# B&R Automation Studio project RobotNewEra (part 9)

#### gmciplog.cnc
```
Root (LangModule=ailgcode, Version=1.0)
  AxesSpec
  PVMacros:
    DR8:
      REF = #next_motion.Data.R8_value
    DI4:
      REF = #next_motion.Data.I4_value
    DU4:
      REF = #next_motion.Data.UI4_value
    DR8_G211:
      SET = %_CNC.TA = ${EXPR};
       if (%_CNC.TA < 0)
         %_CNC.TA = 0;
       endif
        #next_motion.Data.R8_value = ${EXPR};
    Dlp:
      REF = #next_motion.Data.LinMovement.Position
    Dli:
      SET = #next_motion.Data.LinMovement.Idx[0] = ArrayRep(:(:-1:):);
        #next_motion.Data.LinMovement.Idx = ${EXPR};
    Dlm:
      SET = #next_motion.Data.LinMovement.Mode[0] = ArrayRep(:(:-1:):);
        #next_motion.Data.LinMovement.Mode = ${EXPR};
    Dto:
      REF = #next_motion.Data.Trans.Offset
    Dti:
      SET = #next_motion.Data.Trans.AxIdx[0] = ArrayRep(:(:-1:):);
        #next_motion.Data.Trans.AxIdx = ${EXPR};
    Dtm:
      SET = #next_motion.Data.Trans.Mode[0] = ArrayRep(:(:-1:):);
        #next_motion.Data.Trans.Mode = ${EXPR};
    Dcp:
      REF = #next_motion.Data.CircMovement.Parameter
    Dci:
      SET = #next_motion.Data.CircMovement.Idx[0] = ArrayRep(:(:-1:):);
        #next_motion.Data.CircMovement.Idx = ${EXPR};
    Dcm:
      SET = #next_motion.Data.CircMovement.Mode[0] = ArrayRep(:(:-1:):);
        #next_motion.Data.CircMovement.Mode = ${EXPR};
    Dtp:
      REF = #next_motion.Data.ToolAxOrient.Parameter
    Dts:
      REF = #next_motion.Data.ToolAxOrient.Sign
    Daz:
      REF = #next_motion.Data.AbsZeroPtShift.ZpRecIdx
    Dpt:
      SET = #next_motion.Data.ProgZeroPtShift.Type[0] = ArrayRep(:(:-1:):);
        #next_motion.Data.ProgZeroPtShift.Type = ${EXPR};
    Dpm:
      SET = #next_motion.Data.ProgZeroPtShift.Mode[0] = ArrayRep(:(:-1:):);
        #next_motion.Data.ProgZeroPtShift.Mode = ${EXPR};
    Dpa:
      REF = #next_motion.Data.ProgZeroPtShift.AxShift
    Dovpathdef:
      REF = #next_motion.Data.OptMotPar.path_definition
    Dovpathdefd:
      REF = #next_motion.Data.OptMotPar.path_definition_def
    Dorpar:
      REF = #next_motion.Data.OptMotPar.robot_par
    Dorpard:
      REF = #next_motion.Data.OptMotPar.robot_par_def
    Dolim:
      REF = #next_motion.Data.OptMotPar.limits_idx
    Dolimd:
      REF = #next_motion.Data.OptMotPar.limits_idx_def
    Dolimfac:
      REF = #next_motion.Data.OptMotPar.limits_factor
    Dolimfacd:
      REF = #next_motion.Data.OptMotPar.limits_factor_def
    Dfdx:
      REF = #next_motion.Data.FullTrfTool.Dx
    Dfdy:
      REF = #next_motion.Data.FullTrfTool.Dy
    Dfdz:
      REF = #next_motion.Data.FullTrfTool.Dz
    Dfph:
      REF = #next_motion.Data.FullTrfTool.Phi
    Dft:
      REF = #next_motion.Data.FullTrfTool.Theta
    Dfps:
      REF = #next_motion.Data.FullTrfTool.Psi
    DPLDli:
      REF = #next_motion.Data.PosLatchDistance.LatchIdx
    DPLDts:
      REF = #next_motion.Data.PosLatchDistance.TriggSource
    DPLDe:
      REF = #next_motion.Data.PosLatchDistance.Edge
    DPLDti:
      REF = #next_motion.Data.PosLatchDistance.HwTrigIdx
    DPLDd:
      REF = #next_motion.Data.PosLatchDistance.Distance
    DPLli:
      REF = #next_motion.Data.PosLatch.LatchIdx
    DPLts:
      REF = #next_motion.Data.PosLatch.TriggSource
    DPLe:
      REF = #next_motion.Data.PosLatch.Edge
    DPLti:
      REF = #next_motion.Data.PosLatch.HwTrigIdx
    Drma:
      REF = #next_motion.Data.R_DependFeed.MaxRadius
    Drmi:
      REF = #next_motion.Data.R_DependFeed.MinRadius
    Drr:
      REF = #next_motion.Data.R_DependFeed.Rate
    Dsvp:
      SET = #next_motion.Data.Set_v_jump.programmed[0] = ArrayRep(:(:ncOFF:):);
        #next_motion.Data.Set_v_jump.programmed = ${EXPR};
    Dsvv:
      REF = #next_motion.Data.Set_v_jump.value
    Dsap:
      SET = #next_motion.Data.Set_a_jump.programmed[0] = ArrayRep(:(:ncOFF:):);
        #next_motion.Data.Set_a_jump.programmed = ${EXPR};
    Dsav:
      REF = #next_motion.Data.Set_a_jump.value
    Dsep:
      SET = #next_motion.Data.SetAxLimit.programmed[0] = ArrayRep(:(:ncOFF:):);
        #next_motion.Data.SetAxLimit.programmed = ${EXPR};
    Dser:
      REF = #next_motion.Data.SetAxLimit.RecordIdx
    Dcad:
      REF = #next_motion.Data.CamWrapping.Diameter
    Dcap:
      REF = #next_motion.Data.CamWrapping.ParameterP1
    Dsu:
      REF = #next_motion.Data.SetPathAccDec.UnitType
    Dsv108:
      SET = #next_motion.Data.SetPathAccDec.value = ${EXPR};
        if (#next_motion.Data.SetPathAccDec.UnitType == 1)
          %_CNC.lim_path_acc_p = ${EXPR} / 100.0 * %_CNC.lim_path_acc_p_ini;
        else
          %_CNC.lim_path_acc_p = ${EXPR};
        endif
    Dsv109:
      SET = #next_motion.Data.SetPathAccDec.value = ${EXPR};
        if (#next_motion.Data.SetPathAccDec.UnitType == 1)
          %_CNC.lim_path_acc_n = ${EXPR} / 100.0 * %_CNC.lim_path_acc_n_ini;
        else
          %_CNC.lim_path_acc_n = ${EXPR};
        endif
    Dsv110:
      SET = #next_motion.Data.SetPathAccDec.value = ${EXPR};
        if (#next_motion.Data.SetPathAccDec.UnitType == 1)
          %_CNC.lim_path_acc_p = ${EXPR} / 100.0 * %_CNC.lim_path_acc_p_ini;
          %_CNC.lim_path_acc_n = ${EXPR} / 100.0 * %_CNC.lim_path_acc_n_ini;
        else
          %_CNC.lim_path_acc_p = ${EXPR};
          %_CNC.lim_path_acc_n = ${EXPR};
        endif
    Dsma:
      REF = #next_motion.Data.SetTransSpeed.MaxAngle
    Dsmi:
      REF = #next_motion.Data.SetTransSpeed.MinAngle
    Dsr:
      REF = #next_motion.Data.SetTransSpeed.RedFactor
    Dbrp:
      REF = #next_motion.Data.BezierSpline.RadiusProgrammed
    Dbr:
      REF = #next_motion.Data.BezierSpline.Radius
    Dbvp:
      REF = #next_motion.Data.BezierSpline.VeProgrammed
    Dbv:
      REF = #next_motion.Data.BezierSpline.Ve
    Dbl:
      REF = #next_motion.Data.BezierSpline.LinProgrammed
    Dbsf:
      REF = #next_motion.Data.BezierSpline.scalingFactor
    Dbsfd:
      REF = #next_motion.Data.BezierSpline.scalingFactor_def
    Dao:
      REF = #next_motion.Data.AutomTangentialAx.Offset
    Daa:
      REF = #next_motion.Data.AutomTangentialAx.AxIdx
    DAMa:
      REF = #next_motion.Data.AxisMapping.AxIdx
    DAMf:
      REF = #next_motion.Data.AxisMapping.factor
    DAMp:
      REF = #next_motion.Data.AxisMapping.ParameterP1
    DSPEt:
      REF = #next_motion.Data.SignalPathEnd.Time
    DSPEst:
      REF = #next_motion.Data.SignalPathEnd.SignalType
    DSPEsi:
      REF = #next_motion.Data.SignalPathEnd.SignalIdx
    DSPEsd:
      REF = #next_motion.Data.SignalPathEnd.SourceData
    DSPEd:
      REF = #next_motion.Data.SignalPathEnd.DataLength
    DSPEp:
      SET = #next_motion.Data.SignalPathEnd.pDestination = \#sys_vars.EXF[0];
    DSPEDst:
      REF = #next_motion.Data.SignalPathEndDist.SignalType
    DSPEDsi:
      REF = #next_motion.Data.SignalPathEndDist.SignalIdx
    DSPEDsd:
      REF = #next_motion.Data.SignalPathEndDist.SourceData
    DSPEDd:
      REF = #next_motion.Data.SignalPathEndDist.DataLength
    DSPEDp:
      SET = #next_motion.Data.SignalPathEndDist.pDestination = \#sys_vars.EXF[0];
    DSPo:
      REF = #next_motion.Data.SignalPredict.Override
    DWCx1:
      REF = #next_motion.Data.WS_Ctrl.x1
    DWCz1:
      REF = #next_motion.Data.WS_Ctrl.z1
    DWCy1:
      REF = #next_motion.Data.WS_Ctrl.y1
    DWCx2:
      REF = #next_motion.Data.WS_Ctrl.x2
    DWCz2:
      REF = #next_motion.Data.WS_Ctrl.y2
    DWCy2:
      REF = #next_motion.Data.WS_Ctrl.z2
    DWCi:
      REF = #next_motion.Data.WS_Ctrl.index
    DWCc:
      REF = #next_motion.Data.WS_Ctrl.coord
    DWCp:
      REF = #next_motion.Data.WS_Ctrl.pplane
    DWCo:
      REF = #next_motion.Data.WS_Ctrl.orient
    DWCs:
      REF = #next_motion.Data.WS_Ctrl.shape
    DWCa:
      SET = #next_motion.Data.WS_Ctrl.arm_diameter[0] = ArrayRep(:(:ncOFF:):);
        #next_motion.Data.WS_Ctrl.arm_diameter = ${EXPR};
    DTDRt:
      REF = #next_motion.Data.ToolDataRecord.ToolIdx
    Sz:
      REF = #sys_vars.ZP
    DSSi:
      REF = #next_motion.Data.SpindleSpeed.Idx
    DSSs:
      REF = #next_motion.Data.SpindleSpeed.speed
    DCSSt:
      REF = #next_motion.Data.C2_SplineStart.BCType
    DCSSv:
      REF = #next_motion.Data.C2_SplineStart.BCValue
    DCSSp:
      SET = #next_motion.Data.C2_SplineStart.BCProgrammed[0] = ArrayRep(:(:ncOFF:):);
        #next_motion.Data.C2_SplineStart.BCProgrammed = ${EXPR};
    DCSSsp:
      REF = #next_motion.Data.C2_SplineStart.SegmentParameter
    DCSSst:
      REF = #next_motion.Data.C2_SplineStart.SegmentType
    DCSEt:
      REF = #next_motion.Data.C2_SplineEnd.BCType
    DCSEv:
      REF = #next_motion.Data.C2_SplineEnd.BCValue
    DCSEp:
      SET = #next_motion.Data.C2_SplineEnd.BCProgrammed[0] = ArrayRep(:(:ncOFF:):);
        #next_motion.Data.C2_SplineEnd.BCProgrammed = ${EXPR};
    DFd:
      REF = #next_motion.Data.Frame.Data
    DSVs:
      REF = #next_motion.Data.SystemVariable.SysVarIdx
    DSVa:
      REF = #next_motion.Data.SystemVariable.AxIdx
    DSVd:
      REF = #next_motion.Data.SystemVariable.Data.R8_value
    DABNf:
      REF = #next_motion.Data.AutoBlockNumber.offset
    DABNo:
      REF = #next_motion.Data.AutoBlockNumber.factor
    DCSSPs:
      REF = #next_motion.Data.ConstantSurfaceSpeed.Speed
    DCSSPp:
      REF = #next_motion.Data.ConstantSurfaceSpeed.Programmed
    MXFPx:
      REF = #next_motion.Data.MXFrame.Pos.x
    MXFPy:
      REF = #next_motion.Data.MXFrame.Pos.y
    MXFPz:
      REF = #next_motion.Data.MXFrame.Pos.z
    MXFOt:
      REF = #next_motion.Data.MXFrame.Orient.Type
    MXFOa:
      REF = #next_motion.Data.MXFrame.Orient.Angle
    MXTFPx:
      REF = #next_motion.Data.MXTool.Frame.Pos.x
    MXTFPy:
      REF = #next_motion.Data.MXTool.Frame.Pos.y
    MXTFPz:
      REF = #next_motion.Data.MXTool.Frame.Pos.z
    MXTFOt:
      REF = #next_motion.Data.MXTool.Frame.Orient.Type
    MXTFOa:
      REF = #next_motion.Data.MXTool.Frame.Orient.Angle
    MXTr:
      REF = #next_motion.Data.MXTool.Radius
    MXPPx:
      REF = #next_motion.Data.MXPoint.Pos.x
    MXPPy:
      REF = #next_motion.Data.MXPoint.Pos.y
    MXPPz:
      REF = #next_motion.Data.MXPoint.Pos.z
    MXPOt:
      REF = #next_motion.Data.MXPoint.Orient.Type
    MXPOa:
      REF = #next_motion.Data.MXPoint.Orient.Angle
    MXPCm:
      REF = #next_motion.Data.MXPoint.Cfg.Mode
    MXPr:
      REF = #next_motion.Data.MXPoint.RotAxis
    MXPa:
      REF = #next_motion.Data.MXPoint.AuxAxis
    MXPhTr:
      REF = #next_motion.Data.MXPathDesc.Trans.Radius
    MXPhTt:
      REF = #next_motion.Data.MXPathDesc.Trans.Type
    MXDa:
      REF = #next_motion.Data.MXDynamicDesc.Accel
    MXDd:
      REF = #next_motion.Data.MXDynamicDesc.Decel
    MXDOe:
      REF = #next_motion.Data.MXDynamicDesc.Optmot.Enable
    MXDOv:
      REF = #next_motion.Data.MXDynamicDesc.Optmot.VelPathDef
    MXDOr:
      REF = #next_motion.Data.MXDynamicDesc.Optmot.RobotPar
    MXDOl:
      REF = #next_motion.Data.MXDynamicDesc.Optmot.Limits
    MXVv:
      REF = #next_motion.Data.MXVelocity.v
    MXVm:
      REF = #next_motion.Data.MXVelocity.Mode
    MXAj:
      REF = #next_motion.Data.MXAxisTarget.JointAxis
    MXAa:
      REF = #next_motion.Data.MXAxisTarget.AuxAxis
    MXAb:
      REF = #next_motion.Data.MXAxisTarget.BaseAxis
    MXJ:
      REF = #next_motion.Data.MXJointAxis
    MXAto:
      REF = #next_motion.Data.MXAutoTang.Offset
    MXCDCas:
      REF = #next_motion.Data.MXCDC.ArcTransSpd
    MXCDCsm:
      REF = #next_motion.Data.MXCDC.SpdMode
    MXCDCcv:
      REF = #next_motion.Data.MXCDC.ContourViolation
    MXCDCtm:
      REF = #next_motion.Data.MXCDC.TransMode
    MXCDCem:
      REF = #next_motion.Data.MXCDC.EntryMode
    MXCDCal:
      REF = #next_motion.Data.MXCDC.AcrToLine
    THCp:
      REF = #next_motion.Data.ThreadCut.Position
    THCi:
      SET = #next_motion.Data.ThreadCut.Idx[0] = ArrayRep(:(:-1:):);
        #next_motion.Data.ThreadCut.Idx = ${EXPR};
    THCm:
      SET = #next_motion.Data.ThreadCut.Mode[0] = ArrayRep(:(:-1:):);
        #next_motion.Data.ThreadCut.Mode = ${EXPR};
    THCld:
      REF = #next_motion.Data.ThreadCut.LeadDirection
    THCl:
      REF = #next_motion.Data.ThreadCut.Lead
    THCo:
      REF = #next_motion.Data.ThreadCut.Offset
    ACVc:
      REF = #next_motion.Data.AxisCtrlVelocity.Command
    ACVi:
      REF = #next_motion.Data.AxisCtrlVelocity.Idx
    ACSs:
      REF = #next_motion.Data.AxisCtrlSpeed.Speed
    ACSi:
      REF = #next_motion.Data.AxisCtrlSpeed.Idx
    ACPp:
      REF = #next_motion.Data.AxisCtrlPosition.Position
    ACPd:
      REF = #next_motion.Data.AxisCtrlPosition.PositionDefined
    ACPi:
      REF = #next_motion.Data.AxisCtrlPosition.Idx
    ACPm:
      REF = #next_motion.Data.AxisCtrlPosition.Mode
    CHFm:
      REF = #next_motion.Data.Champfer.Mode
    CHFv:
      REF = #next_motion.Data.Champfer.Value
    GENd:
      REF = #next_motion.Data.GenericData.Data
  Constants:
    PathBusy = BUSY (type=STRING)
    PathStatus = STATUS (type=STRING)
    PathErrLevel = ERRLEV (type=STRING)
  BuiltInProcs:
    SendCommand = SendCommand(:$[1]:); (MinArgs=1, MaxArgs=1, Inline=Yes)
    DispatchAndWait = DispatchAndWait(:$[1]:); (MinArgs=1, MaxArgs=1, Inline=Yes)
  Preprocess:
    MP_PJN (Search=MP22000 , Replace=PJN )
    MP_PJB (Search=MP22100 , Replace=PJB )
  GCodes:
    G_DELAY (GNum=0, Alias=@, AliasIsPattern=Yes, Inline=Yes)
      Arg (DataType=FLOAT, ref=tickdelay)
    G_PJN (GNum=22000, Alias=PJN, Inline=Yes, Group=220)
      Arg PathBusy (DataType=FLOAT, ref=busy_count)
      Arg PathStatus (DataType=FLOAT, ref=final_status)
      Arg PathErrLevel (DataType=FLOAT, ref=error_level)
    G_PJB (GNum=22100, Alias=PJB, Inline=Yes, Group=220)
      Arg PathBusy (DataType=FLOAT, ref=busy_count)
      Arg PathStatus (DataType=FLOAT, ref=final_status)
      Arg PathErrLevel (DataType=FLOAT, ref=error_level)
  MCodes:
    M_DEFAULT (IsDefault=Yes, MinValue=0, MaxValue=999999)
      ARG (ref=VALUE, DataType=FLOAT, RequireLiteral=Yes)
    M10003 = 10003 (Inline=Yes)
      ARG (ref=VALUE, DataType=FLOAT, RequireLiteral=Yes)
    M1000000 = 1000000 (Alias=;, AliasIsPattern=Yes, Inline=Yes, IgnoreIfGroups=220)
      ARG (ref=VALUE, DataType=FLOAT, RequireLiteral=Yes)
  ParserData (NestedComments=No, DefaultCaseSensitive=Yes, CommentsSpanLines=No, ReadWholeFileBeforeParsing=No, ExpectMainProgStmts=Yes, UseFubTemplates=No)
    TKG_END_OF_LINE = \n (IsPattern=No)
    TKG_OPEN_COMMENT = #
    TKG_NC_BLOCK_PREFIX = N:[\s\d] (IsPattern=Yes)
    TKG_OPEN_LISTBRACKET = (
    TKG_CLOSE_LISTBRACKET = )
    TKG_COMMA = ,
    TKG_NUMBER = \d+\.\d+|\d+\.|\.\d+ (IsPattern=Yes)
    TKG_INTEGER = \d+ (IsPattern=Yes)
    TKG_NUMBER_EXP = e:[\s\d\+\-\.] (IsPattern=Yes)
    TKG_ASSIGN_EQ = =
    TKG_ARITH_BINARY_MINUS = -
    TKG_M_CODE_PREFIX = MP:\d (IsPattern=Yes)
  StringChars (AsciiStringStart=")
    EscapeSeq (Search=$N, CaseSensitive=No, ReplaceValue=10)
    EscapeSeq (Search=$L, CaseSensitive=Yes, ReplaceValue=10)
    EscapeSeq (Search=$Q, CaseSensitive=No, ReplaceStr=")
    EscapeSeq (Search=$[\dA-F]+, IsPattern=Yes, CaseSensitive=No, ReplaceEncodingBase=16)
    EscapeSeq (Search=$$, ReplaceStr=$)
    EscapeSeq (Search=$, ReplaceStr=)
```

- Data object Logical/MotionHandling/Interpreter/GmcIpConfig/gmcipesm (Cnc, version 2.47.4) (no source held here)

### Data object Logical/MotionHandling/Interpreter/GmcIpConfig/gmcipmxd (Cnc, version 2.47.4)

#### gmcipmxd.cnc
```
(********************************************************************
 * COPYRIGHT -- Bernecker + Rainer
 ********************************************************************
 * Library: Motion Command Extension
 * File: arnc0mx.typ
 * Author: B&R
 ********************************************************************
 * Data types of Motion Command Library
 ********************************************************************)

TYPE
	MXOrientationType : STRUCT
		Type : UDINT;
		Angle : ARRAY[0..3]OF LREAL;
	END_STRUCT;
	MXPositionType : STRUCT
		x : LREAL;
		y : LREAL;
		z : LREAL;
	END_STRUCT;
	MXFrameType : 	STRUCT
		Pos : MXPositionType;
		Orient : MXOrientationType;
	END_STRUCT;
	MXToolType : STRUCT
		Frame : MXFrameType;
		Radius : LREAL;
	END_STRUCT;
	MXJointAxisType :ARRAY[0..5]OF LREAL;
	MXAuxAxisType :ARRAY[0..14]OF LREAL;
	MXBaseAxisType :ARRAY[0..5]OF LREAL;
	MXRotAxisType :ARRAY[0..5]OF LREAL;
	MXConfigType : 	STRUCT
		Mode : UDINT;
	END_STRUCT;
	MXPointType : 	STRUCT
		Pos : MXPositionType;
		Orient : MXOrientationType;
		Cfg : MXConfigType;
		RotAxis : MXRotAxisType;
		AuxAxis : MXAuxAxisType;
	END_STRUCT;
	MXPathTransType : STRUCT
		Radius	:	LREAL;
		Type	:	UDINT;
	END_STRUCT;
	MXPathDescType : STRUCT
		Trans	:	MXPathTransType;
	END_STRUCT;
	MXOptMotType : STRUCT
		Enable : BOOL;
		VelPathDef : USINT;
		RobotPar : USINT;
		Limits : USINT;
	END_STRUCT;
	MXDynamicDescType :	STRUCT
		Accel : LREAL := 100;
		Decel : LREAL := 100;
		Optmot : MXOptMotType;
	END_STRUCT;
	MXHWTrigType : 	STRUCT
		Source : USINT;
		Index : USINT;
	END_STRUCT;
	MXSWTrigType : STRUCT
		Expression : STRING[64];
	END_STRUCT;
	MXTriggConfigType :	STRUCT
		Type : UINT;
		HWTrig : MXHWTrigType;
		SWTrig : MXSWTrigType;
		Edge : USINT;
		ResidPath : USINT;
	END_STRUCT;
	MXVelocityType : STRUCT
		v : LREAL;
		Mode : UDINT := 1;
	END_STRUCT;
	MXAxisTargetType : 	STRUCT
		JointAxis : MXJointAxisType;
		AuxAxis : MXAuxAxisType;
		BaseAxis : MXBaseAxisType;
	END_STRUCT;
	MXCDCType : STRUCT
		ArcTransSpd : LREAL := 100;
		SpdMode : UDINT;
		ContourViolation : UDINT;
		TransMode : UDINT;
		EntryMode : USINT;
		AcrToLine : BOOL;
	END_STRUCT;
	MXAutoTangType : STRUCT
		Offset : LREAL;
	END_STRUCT;
	MXHWTriggerType :	STRUCT
		Source : UINT;
		Index : UINT;
	END_STRUCT;
	MXTriggerConfigType : 	STRUCT
		Type : UINT;
		Edge : UINT;
		HWTrigger : MXHWTriggerType;
	END_STRUCT;
END_TYPE

(********************************************************************
 * COPYRIGHT (C) BERNECKER + RAINER, AUSTRIA, A-5142 EGGELSBERG
 ********************************************************************
 * Library: ARNC0MX
 * File: arnc0mx.fun
 * Created: 13.06.2012
 ********************************************************************
 * Functions and function blocks of library ARNC0MX
 ********************************************************************)
FUNCTION MXPointToJointEx1 : UDINT
	VAR_INPUT
		AddrTrfData : UDINT;
		Point : MXPointType;
		Joint : MXJointAxisType;
		TrfType : UDINT;
		Tool : MXToolType;
		BaseFrame : MXFrameType;
		RefJoint : ARRAY[0..5] OF LREAL;
	END_VAR
END_FUNCTION

FUNCTION MXPointToJointEx : UDINT
	VAR_INPUT
		AddrTrfData : UDINT;
		Point : MXPointType;
		Joint : MXJointAxisType;
		TrfType : UDINT;
		Tool : MXToolType;
		BaseFrame : MXFrameType;
		RefJoint : MXJointAxisType;
	END_VAR
END_FUNCTION

FUNCTION MXJointToPointEx1 : UDINT
	VAR_INPUT
		AddrTrfData : UDINT;
		Joint : MXJointAxisType;
		Point : MXPointType;
		AnglesType : UDINT;
		TrfType : UDINT;
		Tool : MXToolType;
		BaseFrame : MXFrameType;
		RefPath : ARRAY[0..5] OF LREAL;
	END_VAR
END_FUNCTION

FUNCTION MXJointToPointEx : UDINT
	VAR_INPUT
		AddrTrfData : UDINT;
		Joint : MXJointAxisType;
		Point : MXPointType;
		AnglesType : UDINT;
		TrfType : UDINT;
		Tool : MXToolType;
		BaseFrame : MXFrameType;
		RefPoint : MXPointType;
	END_VAR
END_FUNCTION

FUNCTION MXCncAxesToPoint : UDINT
	VAR_INPUT
		AddrTrfData : UDINT;
		Axis : ARRAY[0..14] OF LREAL;
		Point : MXPointType;
		TrfType : UDINT;
		AnglesType : UDINT;
		AxisMapCode : ARRAY[0..14] OF UINT;
		AxisMapIdx : ARRAY[0..14] OF UINT;
		ActiveAxesCount : UDINT;
	END_VAR
END_FUNCTION

FUNCTION MXFromOrient : UDINT
	VAR_INPUT
		Orient : MXOrientationType;
		Matrix : ARRAY[0..8] OF LREAL;
	END_VAR
END_FUNCTION

FUNCTION MXToOrient : UDINT
	VAR_INPUT
		Matrix : ARRAY[0..8] OF LREAL;
		Type : UDINT;
		Orient : MXOrientationType;
		RefAngle : ARRAY[0..2] OF LREAL;
	END_VAR
END_FUNCTION

FUNCTION MXConvertOrient : UDINT
	VAR_INPUT
		OrientIn : MXOrientationType;
		Type : UDINT;
		OrientOut : MXOrientationType;
		RefAngle : ARRAY[0..2] OF LREAL;
	END_VAR
END_FUNCTION

FUNCTION MXFrameRotX : UDINT
	VAR_INPUT
		Frame : MXFrameType;
		Angle : LREAL;
	END_VAR
END_FUNCTION

FUNCTION MXFrameRotY : UDINT
	VAR_INPUT
		Frame : MXFrameType;
		Angle : LREAL;
	END_VAR
END_FUNCTION

FUNCTION MXFrameRotZ : UDINT
	VAR_INPUT
		Frame : MXFrameType;
		Angle : LREAL;
	END_VAR
END_FUNCTION

FUNCTION MXFrameEuler : UDINT
	VAR_INPUT
		Frame : MXFrameType;
		Phi : LREAL;
		Theta : LREAL;
		Psi : LREAL;
	END_VAR
END_FUNCTION

FUNCTION MXFrameRPY : UDINT
	VAR_INPUT
		Frame : MXFrameType;
		Roll : LREAL;
		Pitch : LREAL;
		Yaw : LREAL;
	END_VAR
END_FUNCTION

FUNCTION MXFrameTrans : UDINT
	VAR_INPUT
		Frame : MXFrameType;
		DistanceX : LREAL;
		DistanceY : LREAL;
		DistanceZ : LREAL;
	END_VAR
END_FUNCTION

FUNCTION MXFrameTransX : UDINT
	VAR_INPUT
		Frame : MXFrameType;
		Distance : LREAL;
	END_VAR
END_FUNCTION

FUNCTION MXFrameTransY : UDINT
	VAR_INPUT
		Frame : MXFrameType;
		Distance : LREAL;
	END_VAR
END_FUNCTION

FUNCTION MXFrameTransZ : UDINT
	VAR_INPUT
		Frame : MXFrameType;
		Distance : LREAL;
	END_VAR
END_FUNCTION

FUNCTION MXFrameApply : UDINT
	VAR_INPUT
		Frame1 : MXFrameType;
		Frame2 : MXFrameType;
	END_VAR
END_FUNCTION

FUNCTION MXFromFrame : UDINT
	VAR_INPUT
		Frame : MXFrameType;
		PointIn : MXPointType;
		PointOut : MXPointType;
	END_VAR
END_FUNCTION

FUNCTION MXToFrame : UDINT
	VAR_INPUT
		Frame : MXFrameType;
		PointIn : MXPointType;
		PointOut : MXPointType;
	END_VAR
END_FUNCTION

(********************************************************************
 * COPYRIGHT -- Bernecker + Rainer
 ********************************************************************
 * Library: Motion Command Extension
 * File: arnc0mx.var
 * Author: B&R
 ********************************************************************
 * Constants of Motion Command Library
 ********************************************************************)

(* Velocity mode constants (<MXVelocityType>.Mode) *)
VAR CONSTANT
  MX_VEL_MODE_RAPID : UDINT := 0; (* rapid mode *)
  MX_VEL_MODE_FEED  : UDINT := 1; (* feedrate mode *)
  MX_VEL_MODE_TIME  : UDINT := 2; (* inverse time mode *)
END_VAR

(* MXVelocityType constants *)
VAR CONSTANT
  MX_VEL_RAPID  : MXVelocityType := (Mode:=0);           (* rapid movement         *)
  MX_VEL_F50000 : MXVelocityType := (v:=50000, Mode:=1); (* 50000 units per minute *)
  MX_VEL_F10000 : MXVelocityType := (v:=10000, Mode:=1); (* 10000 units per minute *)
  MX_VEL_F5000  : MXVelocityType := (v:=5000,  Mode:=1); (* 5000 units per minute  *)
  MX_VEL_F1000  : MXVelocityType := (v:=1000,  Mode:=1); (* 1000 units per minute  *)
  MX_VEL_F500   : MXVelocityType := (v:=500,   Mode:=1); (* 500 units per minute   *)
  MX_VEL_F100   : MXVelocityType := (v:=100,   Mode:=1); (* 100 units per minute   *)
END_VAR

(* Trigger configuration constants *)
VAR CONSTANT
  MX_TRIGGER_HW	            : UINT := 0;           (* Hardware trigger - MXHWTriggerType *)
  MX_TRIGGER_POSITIVE_EDGE  : UINT := 0;           (* Positive edge						 *)
  MX_TRIGGER_NEGATIVE_EDGE  : UINT := 1;           (* Negative edge						 *)
  MX_TRIGGER_HW_INPUT1		: UINT := 1;           (* Hardware trigger input 1			 *)
  MX_TRIGGER_HW_INPUT2		: UINT := 2;           (* Hardware trigger input 1			 *)
END_VAR

(* MXFrameMXFrameType constants *)
VAR CONSTANT
  MX_FRM_ZERO : MXFrameType := (0); (* zero (identity) frame *)
END_VAR

(* Transition type constants (<MXPathTransType>.Type) *)
VAR CONSTANT
  MX_TRANS_OFF      : UDINT := 0; (* Transition deactivated *)
  MX_TRANS_ACCURATE : UDINT := 1; (* Accuracy hold *)
  MX_TRANS_ARC      : UDINT := 2; (* Tangential transition arcs *)
  MX_TRANS_ROUND    : UDINT := 3; (* Rounding edges *)
END_VAR

(* Orientation type constants (<MXOrientationType>.Type) matches constants from TRF_LIB *)
VAR CONSTANT
  MX_CARDAN_XYZ_ANGLES    : UDINT := 1;      (* Cardan XYZ angles *)
  MX_EULER_XYZ_ANGLES     : UDINT := 1;      (* Cardan XYZ angles *)
  MX_CARDAN_XZY_ANGLES    : UDINT := 2;      (* Cardan XZY angles *)
  MX_EULER_XZY_ANGLES     : UDINT := 2;      (* Cardan XZY angles *)
  MX_CARDAN_YXZ_ANGLES    : UDINT := 4;      (* Cardan YXZ angles *)
  MX_EULER_YXZ_ANGLES     : UDINT := 4;      (* Cardan YXZ angles *)
  MX_CARDAN_YZX_ANGLES    : UDINT := 8;      (* Cardan YZX angles *)
  MX_EULER_YZX_ANGLES     : UDINT := 8;      (* Cardan YZX angles *)
  MX_CARDAN_ZXY_ANGLES    : UDINT := 16;     (* Cardan ZXY angles *)
  MX_EULER_ZXY_ANGLES     : UDINT := 16;     (* Cardan ZXY angles *)
  MX_CARDAN_ZYX_ANGLES    : UDINT := 32;     (* Cardan ZYX angles *)
  MX_EULER_ZYX_ANGLES     : UDINT := 32;     (* Cardan ZYX angles *)
  MX_EULER_XYX_ANGLES     : UDINT := 64;     (* Euler XYX angles  *)
  MX_EULER_XZX_ANGLES     : UDINT := 128;    (* Euler XZX angles  *)
  MX_EULER_YXY_ANGLES     : UDINT := 256;    (* Euler YXY angles  *)
  MX_EULER_YZY_ANGLES     : UDINT := 512;    (* Euler YZY angles  *)
  MX_EULER_ZXZ_ANGLES     : UDINT := 1024;   (* Euler ZXZ angles  *)
  MX_EULER_ZYZ_ANGLES     : UDINT := 2048;   (* Euler ZYZ angles  *)
  MX_POSITIVE_ANGLES      : UDINT := 4096;   (* mathematically positive angles *)
  MX_NEGATIVE_ANGLES      : UDINT := 8192;   (* mathematically negative angles *)
  MX_DIRECT_ANGLES        : UDINT := 16384;  (* direct "R" rotation matrix     *)
  MX_INDIRECT_ANGLES      : UDINT := 32768;  (* indirect "R^T" rotation matrix *)
  MX_EULER_ANGLES         : UDINT := 1024;   (* Euler ZXZ is commonly in view  *)
  MX_CARDAN_ANGLES        : UDINT := 1;      (* Cardan XYZ is commonly in view *)
  MX_NAUTICAL_ANGLES      : UDINT := 1;      (* Cardan XYZ is commonly in view *)
  MX_TAIT_BRYAN_ANGLES    : UDINT := 1;      (* Cardan XYZ is commonly in view *)
  MX_QUATERNION           : UDINT := 8000;   (* quaternion *)
END_VAR

(* Kinematics configuration mode constants (<MXConfigType>.Mode) matches constants from TRF_LIB *)
VAR CONSTANT
  MX_MODE_FRONT           : UDINT := 1;          (* front *)
  MX_MODE_BACK            : UDINT := 2;          (* back *)
  MX_MODE_CONVEX          : UDINT := 4;          (* convex *)
  MX_MODE_CONCAVE         : UDINT := 8;          (* concave *)
  MX_MODE_POSITIVE        : UDINT := 16;         (* positive *)
  MX_MODE_NEGATIVE        : UDINT := 32;         (* negative *)
  MX_MODE_LEFT            : UDINT := 64;         (* left *)
  MX_MODE_RIGHT           : UDINT := 128;        (* right *)
  MX_MODE_DIRECT          : UDINT := 256;        (* direct *)
  MX_MODE_INDIRECT        : UDINT := 512;        (* indirect *)
  MX_MODE_CONVEX2         : UDINT := 1024;       (* convex2 *)
  MX_MODE_CONCAVE2        : UDINT := 2048;       (* concave2 *)
  MX_MODE_CONVEX3         : UDINT := 4096;       (* convex3 *)
  MX_MODE_CONCAVE3        : UDINT := 8192;       (* concave3 *)
  MX_MODE_HETEROGENEOUS   : UDINT := 16384;      (* heterogeneous *)
  MX_MODE_HOMOGENEOUS     : UDINT := 32768;      (* homogeneous *)
  MX_MODE_LEFT2           : UDINT := 65536;      (* left2 *)
  MX_MODE_RIGHT2          : UDINT := 131072;     (* right2 *)
  MX_MODE_NEG_DIR         : UDINT := 268435456;  (* negative direction forced *)
  MX_MODE_POS_DIR         : UDINT := 536870912;  (* positive direction forced *)
  MX_MODE_IN_SW_ENDS      : UDINT := 1073741824; (* in SW ends *)
END_VAR

(* Cutter diameter compensation constants *)
VAR CONSTANT
  MX_CDC_LEFT                    : UDINT := 0;      (* CDC left *)
  MX_CDC_RIGHT                   : UDINT := 1;      (* CDC right *)
  MX_CDC_SPD_ON_CONTOUR          : UDINT := 0;      (* Path speed moves to the contour *)
  MX_CDC_SPD_ON_TCP              : UDINT := 1;      (* Path speed moves to the center of the tool *)
  MX_CDC_NO_COUNTER_VIOLATION    : UDINT := 0;      (* Do NOT allow contour violations due to very short path *)
  MX_CDC_VIOLATION_SHORT_PATH    : UDINT := 1;      (* Allow contour violations due to very short path sections *)
  MX_CDC_VIOLATION_INNER_EDGE    : UDINT := 2;      (* Allow contour violations due to an inner edge without intersection *)
  MX_CDC_LINEAR_TRANSITION       : UDINT := 0;      (* CDC with linear transitions *)
  MX_CDC_ARC_TRANSITION          : UDINT := 1;      (* CDC with arc transitions *)
  MX_CDC_ENTRY_BLOCK             : UDINT := 0;      (* Activate/deactivate CDC indirectly with transi-tion block *)
  MX_CDC_ENTRY_DIRECT            : UDINT := 1;      (* Activate/deactivate CDC directly *)
  MX_CDC_ENTRY_INDIRECT          : UDINT := 2;      (* Activate/deactivate CDC indirectly *)
  MX_CDC_NO_ARC_TO_LINE          : UDINT := 0;      (* Deactivate replacement of arc with straight line *)
  MX_CDC_ARC_TO_LINE             : UDINT := 1;      (* Activate replacement of arc with straight line *)
END_VAR

(* Transformation function types *)
VAR CONSTANT
  MX_TRF_TYPE_INVERSE            : UDINT := 0;      (* TRF_inverse  function *)
  MX_TRF_TYPE_INVERSE2           : UDINT := 1;      (* TRF_inverse2 function *)
  MX_TRF_TYPE_INVERSE3           : UDINT := 2;      (* TRF_inverse3 function *)
  MX_TRF_TYPE_DIRECT             : UDINT := 0;      (* TRF_direct   function *)
  MX_TRF_TYPE_DIRECT2            : UDINT := 1;      (* TRF_direct2  function *)
  MX_TRF_TYPE_DIRECT3            : UDINT := 2;      (* TRF_direct3  function *)
END_VAR

(* Statuses, warnings, errors *)
VAR CONSTANT
  MX_OK                          : UDINT := 0;     (* Status OK *)
  MX_WARNING_AXES                : UDINT := 2001;  (* Transformation returns valid values with warnings on axes *)
  MX_WARNING_REF_POINT_ANGLES    : UDINT := 2002;  (* Values in reference point or reference joint axes may be ignored due to conversion to another angles type *)
  MX_ERROR_WRONG_ANGLE_TYPE      : UDINT := 6001;  (* Angles type is not supported *)
  MX_ERROR_TRF_DATA_NOT_DEFINED  : UDINT := 6002;  (* Address of the transformation data variable is zero *)
  MX_ERROR_WRONG_ROBOT           : UDINT := 6003;  (* Robot is not supported *)
  MX_ERROR_WRONG_TRF_TYPE        : UDINT := 6004;  (* Transformation type not supported *)
  MX_ERROR_TRF_LIB_NOT_SUPPORTED : UDINT := 6005;  (* Transformation library of not supported version *)
  MX_ERROR_TRF_CMD_CODE			 : UDINT := 8001;  (* Unknown command code *)
  MX_ERROR_TRF_MEASURE           : UDINT := 8002;  (* Unknown measure *)
  MX_ERROR_TRF_ANGLES_TYPE       : UDINT := 8003;  (* Unknown angles type *)
  MX_ERROR_TRF_GEN29_CMD_CODE    : UDINT := 9001;  (* Unknown command code *)
  MX_ERROR_UNKNOWN_ROBOT         : UDINT := 9002;  (* Unknown robot *)
  MX_ERROR_INVALID_TRF_TYPE      : UDINT := 9003;  (* Invalid type of transformation *)
  MX_ERROR_TRF_ERROR_AXES        : UDINT := 10003; (* Transformation function returns error of axis *)
  MX_ERROR_TRF_NOT_LICENSED      : UDINT := 10008; (* Transformation function not licenced *)
  MX_ERROR_TRF_NOT_SUPPORTED     : UDINT := 10009; (* Transformation function not supported *)
  MX_ERROR_FCT_NOT_DEFINED       : UDINT := 10010; (* Transformation function address is zero *)
  MX_ERROR_TRF_INVALID_INPUTS    : UDINT := 10015; (* Invalid inputs for transformation error *)
END_VAR

(* Error offsets *)
VAR CONSTANT
  MX_OFFSET_WARNING              : UDINT := 2000;  (* ARNC0MX warnings *)
  MX_OFFSET_WARNING_TRF_FUN      : UDINT := 4000;  (* TRF_LIB warnings *)
  MX_OFFSET_ERROR                : UDINT := 6000;  (* ARNC0MX errros *)
  MX_OFFSET_ERROR_TRF_FUN        : UDINT := 12000; (* TRF_LIB errors *)
END_VAR

(********************************************************************
 * COPYRIGHT -- Bernecker + Rainer
 ********************************************************************
 * Library: Motion Command Library
 * File: arnc0mxsv.var
 * Author: B&R
 ********************************************************************
 * System Variables of Motion Command Library
 ********************************************************************)
VAR {SHARED_IP_GLOBAL}
   _Frm  : MXFrameType;
   _Tool : MXToolType;
   _Vel  : MXVelocityType;
   _Base : MXFrameType;
   _Ref  : MXJointAxisType;
   _Pth  : MXPathDescType;
   _Dyn  : MXDynamicDescType;
END_VAR

VAR CONSTANT
   FRM_0   : MXFrameType := (0);
   POINT_0 : MXPointType := (0);
   BASE_0  : MXFrameType := (0);
   TOOL_0  : MXToolType  := (0);
   VEL_0   : MXVelocityType := (v:= 10000, Mode:=1); (* Default Feedrate = 10000*)
   REF_0   : MXJointAxisType := (0);
   VEC6_0  : ARRAY[0..5] OF LREAL := 6(0.0);
   PTH_0   : MXPathDescType := (0);
   DYN_0   : MXDynamicDescType := (Optmot:=(Enable:=1));
   AXIS_TARGET_0 : MXAxisTargetType := (0);
END_VAR

VAR {SHARED_IP_GLOBAL}
  __tmp_point : MXPointType;
  __tmp_frame : MXFrameType;
  __tmp_tool : MXToolType;
  __tmp_vel : MXVelocityType;
  __tmp_joint_axis : MXJointAxisType;
  __tmp_axis_target : MXAxisTargetType;
  __tmp_pth : MXPathDescType;
  __tmp_dynamic : MXDynamicDescType;
  __tmp_cdc : MXCDCType;
  __tmp_auto_tang : MXAutoTangType;
  __tmp_trigger : MXTriggerConfigType;
  __mx_status : UDINT;
  __tmp_vec6 : ARRAY[0..5] OF LREAL;
  __tmp_set_pos : ARRAY[0..14] OF LREAL;
  __tmp_axis_code : ARRAY[0..14] OF UINT;
  __tmp_axis_idx : ARRAY[0..14] OF UINT;
END_VAR
```

### Data object Logical/MotionHandling/Interpreter/GmcIpConfig/gmcipmx (Cnc, version 2.47.4)

#### gmcipmx.cnc
```
Root (LangModule=ailgcode, Version=1.0)
  AILHeader = sub OnProgStart
      %_Frm = %FRM_0;
      %_Base = %BASE_0;
      %_Tool = %TOOL_0;
      %_Vel = %VEL_0;
      %_Pth = %PTH_0;
      %_Dyn = %DYN_0;
      BlockCpy(:\%_Ref, \%REF_0:);
    endsub    
    
	sub OnProgEnd
	  #next_motion.Command = MPCMD_SEGMENTATION_END;
      PushPacket(::);
	endsub
  BuiltInProcs:
    WAIT_PP_SYNC = #next_motion.Command = MPCMD_IP_SYNCH_PP;
      PushPacket(::);
      DispatchAndWait(:IPCMD_SYNC_PP_CONT:);
    ERROR_EX = ErrorEx(:"id":$[1],"fmt":$[2],"data":(:$[3],$[4],$[5],$[6],$[7],$[8],$[9],$[10],$[11],$[12],$[13],$[14]:):); (MinArgs=3, MaxArgs=14)
    SET_POINT:
      Arg (ref=POINT, DataType=ANY_DATA, MinCount=1, MaxCount=1)
    SET_TRIGGER_CONFIG:
      Arg (ref=TRIGGER, DataType=ANY_DATA, MinCount=1, MaxCount=1)
      Arg (ref=bHALT, DataType=ANY_DATA, MinCount=1, MaxCount=1)
      Arg (ref=ID, DataType=ANY_DATA, MinCount=1, MaxCount=1)
    SET_WANTED_JOINT:
      Arg (ref=Ref, DataType=ANY_DATA, MinCount=1, MaxCount=1)
    SET_CIRCLE:
      Arg (ref=END_POINT, DataType=ANY_DATA, MinCount=1, MaxCount=1)
      Arg (ref=CIRCLE_POINT, DataType=ANY_DATA, MinCount=1, MaxCount=1)
    SET_AXIS_TARGET:
      Arg (ref=AXIS_TARGET, DataType=ANY_DATA, MinCount=1, MaxCount=1)
    SET_FRAME:
      Arg (ref=Frm, DataType=ANY_DATA, MinCount=0, MaxCount=1)
    SET_BASEFRAME:
      Arg (ref=Base, DataType=ANY_DATA, MinCount=0, MaxCount=1)
    SET_TOOL:
      Arg (ref=Tool, DataType=ANY_DATA, MinCount=0, MaxCount=1)
    SET_PATH_DESC:
      Arg (ref=Pth, DataType=ANY_DATA, MinCount=0, MaxCount=1)
    SET_DYNAMIC_DESC:
      Arg (ref=Dyn, DataType=ANY_DATA, MinCount=0, MaxCount=1)
    SET_VELOCITY:
      Arg (ref=Vel, DataType=ANY_DATA, MinCount=0, MaxCount=1)
    JointToPoint:
      Arg (ref=Joint, UserType=MXJointAxisType, MinCount=1, MaxCount=1)
      Arg (ref=Point, UserType=MXPointType, MinCount=1, MaxCount=1)
    PointToJoint:
      Arg (ref=Point, UserType=MXPointType, MinCount=1, MaxCount=1)
      Arg (ref=Joint, UserType=MXJointAxisType, MinCount=1, MaxCount=1)
    MoveL:
      Arg (ref=POINT, UserType=MXPointType, MinCount=1, MaxCount=1)
      Arg (ref=Frm, UserType=MXFrameType, MinCount=0, MaxCount=1)
      Arg (ref=Base, UserType=MXFrameType, MinCount=0, MaxCount=1)
      Arg (ref=Tool, UserType=MXToolType, MinCount=0, MaxCount=1)
      Arg (ref=Vel, UserType=MXVelocityType, MinCount=0, MaxCount=1)
      Arg (ref=Pth, UserType=MXPathDescType, MinCount=0, MaxCount=1)
      Arg (ref=Dyn, UserType=MXDynamicDescType, MinCount=0, MaxCount=1)
    MoveJ:
      Arg (ref=POINT, UserType=MXPointType, MinCount=1, MaxCount=1)
      Arg (ref=Frm, UserType=MXFrameType, MinCount=0, MaxCount=1)
      Arg (ref=Base, UserType=MXFrameType, MinCount=0, MaxCount=1)
      Arg (ref=Tool, UserType=MXToolType, MinCount=0, MaxCount=1)
      Arg (ref=Vel, UserType=MXVelocityType, MinCount=0, MaxCount=1)
      Arg (ref=Ref, UserType=MXJointAxisType, MinCount=0, MaxCount=1)
      Arg (ref=Pth, UserType=MXPathDescType, MinCount=0, MaxCount=1)
      Arg (ref=Dyn, UserType=MXDynamicDescType, MinCount=0, MaxCount=1)
    MoveC:
      Arg (ref=END_POINT, UserType=MXPointType, MinCount=1, MaxCount=1)
      Arg (ref=CIRCLE_POINT, UserType=MXPointType, MinCount=1, MaxCount=1)
      Arg (ref=Frm, UserType=MXFrameType, MinCount=0, MaxCount=1)
      Arg (ref=Base, UserType=MXFrameType, MinCount=0, MaxCount=1)
      Arg (ref=Tool, UserType=MXToolType, MinCount=0, MaxCount=1)
      Arg (ref=Vel, UserType=MXVelocityType, MinCount=0, MaxCount=1)
      Arg (ref=Pth, UserType=MXPathDescType, MinCount=0, MaxCount=1)
      Arg (ref=Dyn, UserType=MXDynamicDescType, MinCount=0, MaxCount=1)
    MoveA:
      Arg (ref=AXIS_TARGET, UserType=MXAxisTargetType, MinCount=1, MaxCount=1)
      Arg (ref=Vel, UserType=MXVelocityType, MinCount=0, MaxCount=1)
      Arg (ref=Dyn, UserType=MXDynamicDescType, MinCount=0, MaxCount=1)
      Arg (ref=Pth, UserType=MXPathDescType, MinCount=0, MaxCount=1)
    MoveLSearch:
      Arg (ref=POINT, UserType=MXPointType, MinCount=1, MaxCount=1)
      Arg (ref=TRIGGER, UserType=MXTriggerConfigType, MinCount=1, MaxCount=1)
      Arg (ref=bHALT, DataType=IEC_BOOL, MinCount=1, MaxCount=1)
      Arg (ref=ID, DataType=IEC_UINT, MinCount=1, MaxCount=1)
      Arg (ref=Frm, UserType=MXFrameType, MinCount=0, MaxCount=1)
      Arg (ref=Base, UserType=MXFrameType, MinCount=0, MaxCount=1)
      Arg (ref=Tool, UserType=MXToolType, MinCount=0, MaxCount=1)
      Arg (ref=Vel, UserType=MXVelocityType, MinCount=0, MaxCount=1)
      Arg (ref=Pth, UserType=MXPathDescType, MinCount=0, MaxCount=1)
      Arg (ref=Dyn, UserType=MXDynamicDescType, MinCount=0, MaxCount=1)
    WaitTime:
      Arg (ref=set_time, DataType=IEC_LREAL, MinCount=1, MaxCount=1)
    WaitIp = #next_motion.Command = MPCMD_IP_SYNCH;
      if (#restart.playback)
        #next_motion.Data.I4_value = ncSIMULATION;
      else
        #next_motion.Data.I4_value = ncSTANDARD;
      endif
      PushPacket(::);
      DispatchAndWait(:IPCMD_SYNC_PLC_CONT:);
    WaitEndMove = #next_motion.Command = MPCMD_IP_SYNCH_PATH;
      PushPacket(::);
      DispatchAndWait(:IPCMD_SYNC_PATH_CONT:);
    TmpTool = %__tmp_tool.Frame.Pos.x = %_CNC.tool_dx;
      %__tmp_tool.Frame.Pos.y = %_CNC.tool_dy;
      %__tmp_tool.Frame.Pos.z = %_CNC.tool_dz;
      %__tmp_tool.Frame.Orient.Type = %_CNC.tool_angles_type;
      %__tmp_tool.Frame.Orient.Angle[0] = %_CNC.tool_phi;
      %__tmp_tool.Frame.Orient.Angle[1] = %_CNC.tool_theta;
      %__tmp_tool.Frame.Orient.Angle[2] = %_CNC.tool_psi;
      %__tmp_tool.Frame.Orient.Angle[3] = 0;
      %__tmp_tool.Radius = #sys_vars.RAD;
    GetTool:
      Arg (ref=Tool, UserType=MXToolType, MinCount=1, MaxCount=1)
    TmpBaseFrame = %__tmp_frame.Pos.x = %_CNC.base_frame_dx;
      %__tmp_frame.Pos.y = %_CNC.base_frame_dy;
      %__tmp_frame.Pos.z = %_CNC.base_frame_dz;
      %__tmp_frame.Orient.Type = %_CNC.base_frame_angles_type;
      %__tmp_frame.Orient.Angle[0] = %_CNC.base_frame_phi;
      %__tmp_frame.Orient.Angle[1] = %_CNC.base_frame_theta;
      %__tmp_frame.Orient.Angle[2] = %_CNC.base_frame_psi;
      %__tmp_frame.Orient.Angle[3] = 0;
    GetBaseFrame:
      Arg (ref=Frame, UserType=MXFrameType, MinCount=1, MaxCount=1)
    GetJoint:
      Arg (ref=Joint, UserType=MXJointAxisType, MinCount=1, MaxCount=1)
    GetAxisTarget:
      Arg (ref=AxisTarget, UserType=MXAxisTargetType, MinCount=1, MaxCount=1)
    GetLatchPoint:
      Arg (ref=ID, DataType=IEC_UINT, MinCount=1, MaxCount=1)
      Arg (ref=Point, UserType=MXPointType, MinCount=1, MaxCount=1)
      Arg (ref=Event, DataType=IEC_BOOL, MinCount=1, MaxCount=1)
    GetPoint:
      Arg (ref=Point, UserType=MXPointType, MinCount=1, MaxCount=1)
    GetPointIntern = %__tmp_point = %POINT_0;
      
      local $i;
      $i=0;
      lbegin(1)
        %__tmp_axis_code[$i] = %_AX.axis_map[$i];
        %__tmp_axis_idx[$i] = %_AX.axis_map_idx[$i];
        $i = $i + 1;
      lend($i < GetIpInt(:300:))     
      %__mx_status =  MXCncAxesToPoint(:%_CNC.adr_trf_data_mx,  \%__tmp_set_pos, \%__tmp_point,   %_CNC.trf_type, %_CNC.angles_type, \%__tmp_axis_code, \%__tmp_axis_idx, GetIpInt(:300:) :);
      if (%__mx_status > 0)
        
        ErrorEx(:"id":10905,"fmt":"4d4d4d","data":(:GetCurLine(::),4,%__mx_status:):);
      endif
    CDCOn:
      Arg (ref=Direction, DataType=INT, MinCount=1, MaxCount=1)
      Arg (ref=CDC, UserType=MXCDCType, MinCount=0, MaxCount=1)
    CDCOff:
      Arg (ref=CDC, UserType=MXCDCType, MinCount=0, MaxCount=1)
    AutoTangOn:
      Arg (ref=Param, UserType=MXAutoTangType, MinCount=0, MaxCount=1)
    AutoTangOff = #next_motion.Command = MPCMD_MX_TANG_AX_OFF;
      PushPacket(::);
    SetM = local $i, $num_item;
      $i = 1;
      $num_item = ListLength(:${*}:);
      lbegin (1)
        #next_motion.Command = MPCMD_SET_M_FCT;
        #next_motion.Data.I4_value = ListItemValue(:${*}, $i:);  
        PushPacket(::);
        $i = $i + 1;
      lend($i <= $num_item)
      DispatchMPList(::); (MinArgs=1, MaxArgs=10)
  SysVars:
    TRF_DATA_MX $TRF_DATA_MX:
      GET = return %_CNC.adr_trf_data_mx; (ReturnType=IEC_UDINT)
```

### Data object Logical/MotionHandling/Interpreter/GmcIpUserConfig/gmcipvar (Cnc, version 2.47.4)

#### gmcipvar.cnc
```
CONFIG:
  VARIABLES:
    PV = Jog:Jogging.Speed (Alias=JogSpeed, Type=REAL)
    PV = Jog:Jogging.Mode (Alias=JogMode, Type=USINT)
    PV = Jog:Jogging.Step (Alias=JogStep, Type=BOOL, Synch=path_synch)
    PV = Jog:Jogging.MoveAxis (Alias=MoveAxis, Type=SINT, AryDim1=6)
    PV = Jog:Jogging.Run (Alias=JogRun, Type=BOOL, Synch=path_synch)
    PV = Jog:Jogging.Run (Alias=JogLimit, Type=BOOL, Synch=path_syn ch)
```

- Data object Logical/MotionHandling/Interpreter/GmcIpUserConfig/gmcipfun (Cnc, version 2.47.4) (no source held here)

- Data object Logical/MotionHandling/Interpreter/GmcIpUserConfig/gmcipfub (Cnc, version 2.47.4) (no source held here)

- Data object Logical/MotionHandling/Interpreter/GmcIpUserConfig/gmcipubr (Cnc, version 2.47.4) (no source held here)

- Data object Logical/MotionHandling/Interpreter/GmcIpUserConfig/gmcipusm (Cnc, version 2.47.4) (no source held here)

- Data object Logical/MotionHandling/Interpreter/GmcIpUserConfig/gmcipus (Cnc, version 2.47.4) (no source held here)

- Data object Logical/MotionHandling/Interpreter/GmcIpUserConfig/gmcipuc (Cnc, version 2.47.4) (no source held here)

### Package Logical/MotionHandling/FeedForward - NOT USED

### OptMotConfig.var
```iecst
VAR
	Par6axATrf : ARRAY[0..31] OF TRF_DYN04B_typ := [32(0)];
END_VAR
```

### Program Logical/MotionHandling/FeedForward/6axATrqFF (ANSIC) - Cyclically writes the FF

#### 6axATrqFF.c - Implementation code
```c
/********************************************************************
 * COPYRIGHT -- Bernecker + Rainer
 ********************************************************************
 * Program: 6axATrqFF
 * File: 6axATrqFF.c
 * Author: frigenif
 * Created: May 17, 2011
 ********************************************************************
 * Implementation of program 6axATrqFF
 ********************************************************************/

#include <bur/plctypes.h>

#ifdef _DEFAULT_INCLUDES
 #include <AsDefault.h>
#endif

#include "math.h"

#define PI 	3.1415926535897932384626433832795

void _INIT axATrqFFINIT( void )
{
	TrqFF6axA.Enable = 0;

	TrqFF6axA.Axes[0].Index = AXIS_Q1;
	TrqFF6axA.Axes[0].Sign = 0;				//-1;
	TrqFF6axA.Axes[0].MaxTorque = 6.6;  	//5.5;

	TrqFF6axA.Axes[1].Index = AXIS_Q2;
	TrqFF6axA.Axes[1].Sign = 1;
	TrqFF6axA.Axes[1].MaxTorque = 9.5;		//7.4;

	TrqFF6axA.Axes[2].Index = AXIS_Q3;
	TrqFF6axA.Axes[2].Sign = -1;
	TrqFF6axA.Axes[2].MaxTorque = 6.2;		//3.42;

	TrqFF6axA.Axes[3].Index = AXIS_Q4;
	TrqFF6axA.Axes[3].Sign = -1;
	TrqFF6axA.Axes[3].MaxTorque = 2;	//1.35;

	TrqFF6axA.Axes[4].Index = AXIS_Q5;
	TrqFF6axA.Axes[4].Sign = 1;
	TrqFF6axA.Axes[4].MaxTorque = 1.5;		//0.68;

	TrqFF6axA.Axes[5].Index = AXIS_Q6;
	TrqFF6axA.Axes[5].Sign = -1;
	TrqFF6axA.Axes[5].MaxTorque = 1.5;		//0.68;

	TrqFF6axA.Ramp = 0;

	CncProgWasActive = 0;
	TrqFF6axA.Enable = 0;

}

void _CYCLIC axATrqFFCYCLIC( void )
{

	/*************************** Check if system initialization is completed ***************************/

	if (AxesAddress == 0)
	{
		return;
	}
	else	/* access motion control structures */
	{
		pAxes = (Axes_Type*) AxesAddress;
	}

	AllAxControllerOn = 1;
	AllAxHomingOk = 1;
	for (i=0; i<=5; i++)
	{
		if ((*pAxes)[TrqFF6axA.Axes[i].Index].Output.Status.ControllerStatus != ncTRUE)
		{
			AllAxControllerOn = 0;
		}
		if ((*pAxes)[TrqFF6axA.Axes[i].Index].Output.Status.HomingOk != ncTRUE)
		{
			AllAxHomingOk = 0;
		}
	}

	/*************************** Check if feed forward is active and enabled ***************************/

	OptMotInMotion = 0;
	for (i=0; i<=14; i++)
	{
		/* check if any position != 0 */
		if(OptMotConfig.monitor.s_joint[i] != 0.0)
			OptMotInMotion = 1;
	}

	if(	TrqFF6axA.Enable && AllAxControllerOn && AllAxHomingOk )
	{
		if(OptMotInMotion != 0)
			CncProgWasActive = 1;
		if(CncProgWasActive == 1)
			TrqFF6axA.Active = 1;
		else
			TrqFF6axA.Active = 0;
	}
	else
	{
		CncProgWasActive = 0;
		TrqFF6axA.Active = 0;
	}

	/*************************** ramp FF torque to prevent jumps ***************************/

	if(TrqFF6axA.Active)
	{
		TrqFF6axA.Ramp+=0.005;
		if(TrqFF6axA.Ramp>1.0)
			TrqFF6axA.Ramp=1.0;
	}
	else
	{
		TrqFF6axA.Ramp=0.0;
	}

	/*************************** write FF torque to servo drives ***************************/

	for (i=0; i<6; i++)
	{

		/* skip jumps to zero - except for axis J1 */
		if ((TrqFF6axA.Axes[i].SetTorque !=0) && (OptMotConfig.monitor.feed_forward_torque[6+i] == 0) && (i!=0))
		{
				OptMotConfig.monitor.feed_forward_torque[6+i] = TrqFF6axA.Axes[i].SetTorque;
		}

	//	 filter FF torque
		TrqFF6axA.Axes[i].SetTorque = (REAL) OptMotConfig.monitor.feed_forward_torque[6+i];

		/* limit set torque to motor limits */
		if (TrqFF6axA.Axes[i].SetTorque > TrqFF6axA.Axes[i].MaxTorque)
		{
			TrqFF6axA.Axes[i].SetTorque = TrqFF6axA.Axes[i].MaxTorque;
		}
		else if (TrqFF6axA.Axes[i].SetTorque < -TrqFF6axA.Axes[i].MaxTorque)
		{
			TrqFF6axA.Axes[i].SetTorque = -TrqFF6axA.Axes[i].MaxTorque;
		}

		if(TrqFF6axA.Active)
		{
			TrqFF6axA.Axes[i].CorrectTorque = TrqFF6axA.Axes[i].SetTorque * TrqFF6axA.Axes[i].Sign * TrqFF6axA.Ramp;
			memcpy (&(pAxes[0]+TrqFF6axA.Axes[i].Index)->Input.Parameter.PDOWriteValue[0], &TrqFF6axA.Axes[i].CorrectTorque, 4);
		}
		else
		{
			TrqFF6axA.Axes[i].SetTorque = 0;
			TrqFF6axA.Axes[i].CorrectTorque = 0;
			memcpy (&(pAxes[0]+TrqFF6axA.Axes[i].Index)->Input.Parameter.PDOWriteValue[0], &TrqFF6axA.Axes[i].CorrectTorque, 4);
		}

	}

}
```

#### 6axATrqFF.typ - Local data types
```iecst
(********************************************************************
 * COPYRIGHT -- Bernecker + Rainer
 ********************************************************************
 * Program: 6axATrqFF
 * File: 6axATrqFF.typ
 * Author: frigenif
 * Created: May 17, 2011
 ********************************************************************
 * Local data types of program 6axATrqFF
 ********************************************************************)

TYPE
	TrqFF6axA_Type : 	STRUCT
		Enable : BOOL;
		Axes : ARRAY[0..5] OF TrqFF6axA_Axes_Type;
		Ramp : REAL;
		Active : BOOL;
	END_STRUCT;
	TrqFF6axA_Axes_Type : 	STRUCT
		Index : USINT;
		Sign : REAL;
		MaxTorque : REAL;
		SetTorque : REAL;
		CorrectTorque : REAL;
	END_STRUCT;
END_TYPE
```

#### 6axATrqFF.var - Local variables
```iecst
(********************************************************************
 * COPYRIGHT -- Bernecker + Rainer
 ********************************************************************
 * Program: 6axATrqFF
 * File: 6axATrqFF.var
 * Author: frigenif
 * Created: May 17, 2011
 ********************************************************************
 * Local variables of program 6axATrqFF
 ********************************************************************)
VAR
	AllAxHomingOk : BOOL;
	AllAxControllerOn : BOOL;
	TrqFF6axA : TrqFF6axA_Type;
	pAxes : REFERENCE TO ARRAY[0..MAX_AX_MINUS_ONE] OF Axes_Type;
	i : USINT;
	OptMotInMotion : BOOL;
	CncProgWasActive : BOOL;
	AxesAddress : UDINT := 0;
END_VAR
```

### Package Logical/MotionHandling/Optimizer - Optimizer

### Optimizer.typ - Global data types
```iecst
(********************************************************************
 * COPYRIGHT -- Microsoft
 ********************************************************************
 * Package: Optimizer
 * File: Optimizer.typ
 * Author: renj
 * Created: April 24, 2015
 ********************************************************************
 * Data types of package Optimizer
 ********************************************************************)

TYPE
	ARNC0FILEMONENTRY_typ : 	STRUCT
		name : UDINT; (* File name (address) *)
		path_name : UDINT; (* Full path file name (address) *)
		dir_name : UDINT; (* Directory name (address) *)
		device_name : UDINT; (* Device name (address) *)
		prog_nr : UDINT; (* Number of loaded program *)
		storage_type : UDINT; (* Storage type: 1-file, 2-module *)
		time_stamp : UDINT; (* File time stamp *)
		precompiled_lcf : BOOL; (* Loaded file is laguage configuration file *)
		NOT_USE_1 : ARRAY[0..2]OF USINT;
		next : UDINT; (* Next element in file list *)
	END_STRUCT;
	ARNC0FILEMONBASIC_typ : 	STRUCT
		name : STRING[31]; (* Name of loaded file *)
		prog_nr : UDINT; (* Number of loaded program *)
		storage_type : UDINT; (* Storage type: 1-file, 2-module *)
	END_STRUCT;
	ARNC0FILEMONACCESS_typ : 	STRUCT
		valid : BOOL; (* Extended data can be accessed *)
		NOT_USE_1 : ARRAY[0..2]OF USINT;
		first : UDINT; (* Begin of the file list *)
	END_STRUCT;
	ARNC0FILEMON_typ : 	STRUCT
		set_offset : UDINT; (* Required file offset *)
		offset : UDINT; (* Offset of displayed files *)
		file : ARRAY[0..31]OF ARNC0FILEMONBASIC_typ; (* File monitor *)
		direct_access : ARNC0FILEMONACCESS_typ; (* Access to extended data *)
		handshake : BOOL; (* Set to update data *)
		NOT_USE_1 : ARRAY[0..2]OF USINT;
	END_STRUCT;
	ARNC0EXTWMCOL_typ : 	STRUCT
		result : UDINT; (* WM result *)
		index1 : UDINT; (* Index of 1st found colliding area *)
		shape1 : UDINT; (* Shape of colliding area: 1-block, 2-hspace *)
	END_STRUCT;
	ARNC0EXTWM_typ : 	STRUCT
		joint_position : ARRAY[0..11]OF LREAL; (* Joint coordinate *)
		xyz_position : ARRAY[0..2]OF LREAL; (* TCP position if joints cannot be used *)
		D_FULL : ARRAY[0..5]OF LREAL; (* General tool *)
		local_frame : ARRAY[0..5]OF LREAL; (* Local (base) frame *)
		collision : ARNC0EXTWMCOL_typ; (* Additional information about collisions *)
	END_STRUCT;
	OPTMOT_SEG_CONFIG_typ : 	STRUCT
		distance : LREAL; (* Length of the path segments in CNC units *)
		increase_num_seg_from_radius : LREAL; (* Finer segmentation of circles with smaller radius *)
		increase_num_seg_orient_factor : LREAL; (* Finer segmentation of orientation change *)
		G126_num_seg : UDINT; (* Finer segmentation of rounding edge *)
		G126_num_seg_PTP_Interp : UDINT; (* Finer segmentation of rounding edge *)
	END_STRUCT;
	OPTMOT_AXES_typ : 	STRUCT
		ax_count : UDINT; (* Number of axes for optimization *)
		ax_index : ARRAY[0..14]OF USINT; (* Index of CNC-axis *)
		NOT_USE_1 : USINT;
		ax_factor : ARRAY[0..14]OF LREAL; (* Scaling factor *)
	END_STRUCT;
	OPTMOT_PATHDEF_typ : 	STRUCT
		type : UINT; (* Type of path definition *)
		ax_count : UINT; (* Number of axes for path computation *)
		ax_index : ARRAY[0..14]OF USINT; (* Index of CNC-axis *)
		NOT_USE_1 : USINT;
		ax_factor : ARRAY[0..14]OF LREAL; (* Scaling factor *)
	END_STRUCT;
	OPTMOT_TRF_VAR_INSTANCES_typ : 	STRUCT
		trf_var_ip : UDINT; (* For developers only *)
		trf_var_ip_wm : UDINT; (* For developers only *)
		trf_var_pp1 : UDINT; (* For developers only *)
		trf_var_pp2 : UDINT; (* For developers only *)
		trf_var_bgen : UDINT; (* For developers only *)
	END_STRUCT;
	OPTMOT_ACCESS_POINTS_typ : 	STRUCT
		pp_context : UDINT; (* Access of data for external workspace monitoring *)
		wm_function : UDINT; (* Access for external call of workspace monitoring *)
		address_debug_data : UDINT; (* For developers only *)
		trf_var_instances : OPTMOT_TRF_VAR_INSTANCES_typ; (* Structure of access points for developers only *)
	END_STRUCT;
	OPTMOT_INTERNAL_typ : 	STRUCT
		buffer_nc_block : UDINT; (* Size of a buffer containing NC-blocks *)
		buffer_geometric_data : UDINT; (* Size of a buffer containing geometric data of the path *)
		disable_optmot_for_channel : USINT; (* Deactivation of optimizer for current CNC channel *)
		Ts_multiple : USINT; (* Sample time of trajectory planer *)
		linear_feed : USINT; (* Behavior of path acceleration *)
		bypass_optmot : USINT; (* Simulation mode *)
		addr_dyn_model : UDINT; (* Pointer to the dynamic model *)
		der_num_poly_points : UINT; (* Number of segments used for derivatives computation *)
		geometric_pos_filter : UINT; (* Number of segments used for position filter *)
		buffer_level_lookahead : UINT; (* Minimal fill level of lookahead buffer *)
		G220_reduce_to_max_in_buffer : UINT; (* Reduction of G220 time *)
		sigma_diff_compute : LREAL; (* Lookahead of segmentation *)
		max_angle : LREAL; (* Angle to detect stops on path *)
		access_points : OPTMOT_ACCESS_POINTS_typ; (* Structure of access points for developers only *)
		reserve1 : ARRAY[0..9]OF LREAL; (* For developers only *)
		reserve2 : ARRAY[0..9]OF DINT; (* For developers only *)
	END_STRUCT;
	OPTMOT_LIMITS_typ : 	STRUCT
		v_joint_min : ARRAY[0..14]OF LREAL; (* Minimal velocity limits of the joint axes *)
		v_joint_max : ARRAY[0..14]OF LREAL; (* Maximal velocity limits of the joint axes *)
		a_joint_min : ARRAY[0..14]OF LREAL; (* Minimal acceleration limits of the joint axes *)
		a_joint_max : ARRAY[0..14]OF LREAL; (* Maximal acceleration limits of the joint axes *)
		j_joint_min : ARRAY[0..14]OF LREAL; (* Minimal jerk limits of the joint axes *)
		j_joint_max : ARRAY[0..14]OF LREAL; (* Maximal jerk limits of the joint axes *)
		torque_min : ARRAY[0..14]OF LREAL; (* Minimal torque limits of the joint axes *)
		torque_max : ARRAY[0..14]OF LREAL; (* Maximal torque limits of the joint axes *)
		torque_limits_in_generator_mode : UDINT; (* Activation of generator mode *)
		torque_gen_factor_min : ARRAY[0..14]OF LREAL; (* Factor for minimal torque limit in generator mode *)
		torque_gen_factor_max : ARRAY[0..14]OF LREAL; (* Factor for maximal torque limit in generator mode *)
		v_path_min : ARRAY[0..31]OF LREAL; (* Minimal velocity limits of the path definitions *)
		v_path_max : ARRAY[0..31]OF LREAL; (* Maximal velocity limits of the path definitions *)
		a_path_min : ARRAY[0..31]OF LREAL; (* Minimal acceleration limits of the path definitions *)
		a_path_max : ARRAY[0..31]OF LREAL; (* Maximal acceleration limits of the path definitions *)
		j_path_min : ARRAY[0..31]OF LREAL; (* Minimal jerk limits of the path definitions *)
		j_path_max : ARRAY[0..31]OF LREAL; (* Maximal jerk limits of the path definitions *)
	END_STRUCT;
	OPTMOT_ACTIVE_LIMIT_typ : 	STRUCT
		type : USINT; (* Type of the active limit *)
		source : USINT; (* Source of the active limit *)
		min_max : SINT; (* Positive or negative range of the active limit *)
		index : USINT; (* Index of the axis or path definition of the active limit *)
	END_STRUCT;
	OPTMOT_MONITOR_typ : 	STRUCT
		s_joint : ARRAY[0..14]OF LREAL; (* Cyclical joint position in CNC units *)
		v_joint : ARRAY[0..14]OF LREAL; (* Cyclical joint velocity in CNC units *)
		a_joint : ARRAY[0..14]OF LREAL; (* Cyclical joint acceleration in CNC units *)
		j_joint : ARRAY[0..14]OF LREAL; (* Cyclical joint jerk in CNC units *)
		feed_forward_torque : ARRAY[0..14]OF LREAL; (* Cyclical joint torque/force *)
		v_path : ARRAY[0..31]OF LREAL; (* Cyclical path velocity in CNC units *)
		active_limit : OPTMOT_ACTIVE_LIMIT_typ; (* Structure of information about current limitation *)
		data_valid : UINT; (* Feed forward data is valid *)
		fill_level_lookahead : UINT; (* Fill level of lookahead buffer *)
		reserve : ARRAY[0..1]OF UDINT;
	END_STRUCT;
	OPTMOT_COND_STOP_typ : 	STRUCT
		active : UINT; (* Conditional stop active *)
		call_stop_internal : UINT; (* Internal execution of the conditional stop *)
		identifier : UDINT; (* Identifier of the conditional stop *)
		select_overlapped_identifier : UDINT; (* Selection of identifier in overlapping conditional stops *)
		select_identifier_stop_internal : UDINT; (* Selection of identifier if conditional stop is executed internally *)
	END_STRUCT;
	OPTMOT_COND_STOP_OPTMOT_typ : 	STRUCT
		identifier_aktiv : UDINT; (* Output of aktive identifier *)
		identifier_fulfilled : UDINT; (* Input of fulfilled identifier *)
	END_STRUCT;
	OPTMOT_STOPPING_typ : 	STRUCT
		G126_skip_if_stop : UINT; (* Skip G126 if a stop on path occurs *)
		trajectory : UINT; (* Definition of stopping trajectory *)
		conditional_stop : OPTMOT_COND_STOP_typ; (* Structure of conditional stop *)
		conditional_stop_optmot : OPTMOT_COND_STOP_OPTMOT_typ; (* Structure of optmot synchronal conditional stop *)
	END_STRUCT;
	OPTMOT_PATH_typ : 	STRUCT
		G126_skip_smaller_radius : LREAL; (* Skip G126 if programmed radius is smaller *)
		G126_round_whole_line : UDINT; (* Round whole first/last line *)
		count : UDINT; (* Number of path definitions *)
		definition : ARRAY[0..31]OF OPTMOT_PATHDEF_typ; (* Structure of path definitions parameters *)
		stopping : OPTMOT_STOPPING_typ; (* Structure of stopping parameters *)
		reserve1 : ARRAY[0..170]OF UDINT;
	END_STRUCT;
	OPTMOT_CONFIG_typ : 	STRUCT
		axes : OPTMOT_AXES_typ; (* Structure of joint axes parameters *)
		path : OPTMOT_PATH_typ; (* Structure of path parameters *)
		limits : ARRAY[0..31]OF OPTMOT_LIMITS_typ; (* Structure of limit parameters *)
		segmentation : OPTMOT_SEG_CONFIG_typ; (* Structure of segmentation parameters *)
		monitor : OPTMOT_MONITOR_typ; (* Structure of monitor parameters *)
		internals : OPTMOT_INTERNAL_typ; (* Structure of internal parameters *)
	END_STRUCT;
	OPTMOT_MONITOR_ADVANCED_typ : 	STRUCT
		s_joint : ARRAY[0..14]OF LREAL; (* Cyclical joint position in CNC units *)
		v_joint : ARRAY[0..14]OF LREAL; (* Cyclical joint velocity in CNC units *)
		a_joint : ARRAY[0..14]OF LREAL; (* Cyclical joint acceleration in CNC units *)
		j_joint : ARRAY[0..14]OF LREAL; (* Cyclical joint jerk in CNC units *)
		feed_forward_torque : ARRAY[0..14]OF LREAL; (* Cyclical joint torque/force *)
		v_path : ARRAY[0..31]OF LREAL; (* Cyclical path velocity in CNC units *)
		active_limit : OPTMOT_ACTIVE_LIMIT_typ; (* Structure of information about current limitation *)
		data_valid : UINT; (* Feed forward data is valid *)
		fill_level_lookahead : UINT; (* Fill level of lookahead buffer *)
		tracking_active : UINT; (* Tracking active *)
		tracking_synch : UINT; (* Robot synchronized with conveyor *)
		tracking_index : UINT; (* Active tracking index *)
		reserve : UINT;
	END_STRUCT;
	OPTMOT_TRACKING_ORIENTATION_typ : 	STRUCT
		phi : LREAL; (* Phi-component of a rotation *)
		theta : LREAL; (* Theta-component of a rotation *)
		psi : LREAL; (* Psi-component of a rotation *)
	END_STRUCT;
	OPTMOT_TRACKING_ORIENT_PARAM_typ : 	STRUCT
		measure : UDINT; (* Unit of measurement of the angles *)
		angles_type : UDINT; (* Angles type *)
	END_STRUCT;
	OPTMOT_TRACKING_LIMITS_typ : 	STRUCT
		maxVelocity : LREAL; (* Maximal velocity of the conveyor belt *)
	END_STRUCT;
	OPTMOT_TRACKING_CYCLIC_typ : 	STRUCT
		position : LREAL; (* Cyclical position of the conveyor belt *)
		velocity : LREAL; (* Cyclical velocity of the conveyor belt *)
	END_STRUCT;
	OPTMOT_TRACKING_CONVEYOR_typ : 	STRUCT
		limits : OPTMOT_TRACKING_LIMITS_typ; (* Structure of conveyor limits *)
		orientation : OPTMOT_TRACKING_ORIENTATION_typ; (* Structure of orientation between global basic frame and conveyor belt frame *)
		cyclicData : OPTMOT_TRACKING_CYCLIC_typ; (* Structure of cyclic data *)
	END_STRUCT;
	OPTMOT_TRACKING_CONVEYORDATA_typ : 	STRUCT
		orientationParameter : OPTMOT_TRACKING_ORIENT_PARAM_typ; (* Structure of general orientation parameters *)
		conveyor : ARRAY[0..9]OF OPTMOT_TRACKING_CONVEYOR_typ; (* Structure of conveyor belt data *)
	END_STRUCT;
	OPTMOT_TRACKING_typ : 	STRUCT
		enable : UDINT; (* Enable tracking *)
		conveyorData : OPTMOT_TRACKING_CONVEYORDATA_typ; (* Structure of conveyor belt tracking *)
		reserve1 : ARRAY[0..7]OF LREAL; (* For developers only *)
		reserve2 : ARRAY[0..31]OF UDINT; (* For developers only *)
	END_STRUCT;
	OPTMOT_PATH_ADVANCED_typ : 	STRUCT
		G126_skip_smaller_radius : LREAL; (* Skip G126 if programmed radius is smaller *)
		G126_round_whole_line : UDINT; (* Round whole first/last line *)
		count : UDINT; (* Number of path definitions *)
		definition : ARRAY[0..31]OF OPTMOT_PATHDEF_typ; (* Structure of path definitions parameters *)
		stopping : OPTMOT_STOPPING_typ; (* Structure of stopping parameters *)
		tracking : OPTMOT_TRACKING_typ; (* Structure of tracking parameters *)
	END_STRUCT;
	OPTMOT_CONFIG_ADVANCED_typ : 	STRUCT
		axes : OPTMOT_AXES_typ; (* Structure of joint axes parameters *)
		path : OPTMOT_PATH_ADVANCED_typ; (* Structure of path parameters *)
		limits : ARRAY[0..31]OF OPTMOT_LIMITS_typ; (* Structure of limit parameters *)
		segmentation : OPTMOT_SEG_CONFIG_typ; (* Structure of segmentation parameters *)
		monitor : OPTMOT_MONITOR_ADVANCED_typ; (* Structure of monitor parameters *)
		internals : OPTMOT_INTERNAL_typ; (* Structure of internal parameters *)
	END_STRUCT;
	ARNC0PLOTDATA01_typ : 	STRUCT
		block_ncprog : UDINT; (* Block number *)
		line_ncprog : UDINT; (* Line number *)
		MpId : UDINT; (* Motion packet ident *)
		MpSubId : UDINT; (* Motion packet subident *)
		cmd_code : UINT; (* Command *)
		reserve : UINT; (* don't use *)
		data : ARRAY[0..51]OF USINT; (* Data *)
	END_STRUCT;
	ARNC0PLOTDATA02_typ : 	STRUCT
		block_ncprog : UDINT; (* Block number *)
		line_ncprog : UDINT; (* Line number *)
		MpId : UDINT; (* Motion packet ident *)
		MpSubId : UDINT; (* Motion packet subident *)
		cmd_code : UINT; (* Command *)
		reserve : UINT; (* don't use *)
		data : ARRAY[0..51]OF USINT; (* Data *)
	END_STRUCT;
	ARNC0PLDMOVE_typ : 	STRUCT
		ep : ARRAY[0..2]OF REAL; (* End point *)
		cp : ARRAY[0..2]OF REAL; (* Center point *)
		radius : REAL; (* Tool radius *)
		v_ncprog : REAL; (* Programmed feedrate *)
		info : UDINT; (* Info bits *)
	END_STRUCT;
	ARNC0PLDMOVE02_typ : 	STRUCT
		ep : ARRAY[0..2]OF REAL; (* End point *)
		cp : ARRAY[0..2]OF REAL; (* Center point *)
		radius : REAL; (* Tool radius *)
		v_ncprog : REAL; (* Programmed feedrate *)
		t : REAL; (* block runtime *)
		s : REAL; (* block length, interpolated axes *)
		s_all : REAL; (* block length, all axes *)
		info : UDINT; (* Info bits *)
	END_STRUCT;
	ARNC0PLDPROGEND_typ : 	STRUCT
		t : REAL; (* estimated runtime *)
		s : REAL; (* path length, interpolated axes *)
		s_all : REAL; (* path length, all axes *)
	END_STRUCT;
	ARNC0PLDPROGSTART_typ : 	STRUCT
		ProgNumber : UDINT; (* program number *)
	END_STRUCT;
	ARNC0PLDTOOL_typ : 	STRUCT
		radius : REAL; (* Tool radius *)
		length : REAL; (* Tool length *)
		offset : ARRAY[0..2]OF REAL; (* Tool offset *)
		index : UINT; (* Tool index, tool data number *)
		reserve : UINT; (* don't use *)
	END_STRUCT;
	ARNC0PLDCSTRF_typ : 	STRUCT
		matrix : ARRAY[0..8]OF REAL; (* Rotation matrix *)
		offset : ARRAY[0..2]OF REAL; (* Offset (cs + tool) *)
		info : UDINT; (* Info bits *)
	END_STRUCT;
	ARNC0PLDUSER_typ : 	STRUCT
		data : ARRAY[0..51]OF USINT; (* User data *)
	END_STRUCT;
	ARNC0TRFIODATA_typ : 	STRUCT
		status : UDINT; (* Return status of the last call of the transformation function *)
		in_pos : ARRAY[0..11]OF LREAL; (* Input positions of the transformation function *)
		in_pos_ext : ARRAY[0..11]OF LREAL; (* Extended input positions of the transformation function *)
		out_pos : ARRAY[0..71]OF LREAL; (* Output positions of the transformation function *)
		info : ARRAY[0..8]OF UDINT; (* Information about the last call of the transformation function *)
	END_STRUCT;
	ARNC0WSCTRL_typ : 	STRUCT
		link_index : UDINT; (* index of colliding link *)
		link2_index : UDINT; (* index of colliding link for self-collision *)
		area_index : UDINT; (* index of colliding area *)
	END_STRUCT;
	ARNC0IP_MON_typ : 	STRUCT
		enable : USINT; (*Enable cyclic update *)
		reserve : ARRAY[0..2]OF USINT; (*[RESERVE] *)
		status_msg : ARRAY[0..79]OF USINT; (*String: current status of interpreter e.g. Running/Waiting/Finished *)
		last_error_msg : ARRAY[0..119]OF USINT; (*String: last error message issued *)
		last_error_code : UINT; (*Last status message code issued *)
		loaded_prog_count : UINT; (*Number of files loaded *)
		prog_name : ARRAY[0..79]OF USINT; (*Name of start-program *)
		ncblock_l2 : ARRAY[0..79]OF USINT; (*Interpeter block monitor: current line -2 *)
		ncblock_l1 : ARRAY[0..79]OF USINT; (*Interpeter block monitor: current line -1 *)
		ncblock : ARRAY[0..79]OF USINT; (*Interpeter block monitor: current line *)
		ncblock_n1 : ARRAY[0..79]OF USINT; (*Interpeter block monitor: current line +1 *)
		ncblock_n2 : ARRAY[0..79]OF USINT; (*Interpeter block monitor: current line +2 *)
		cur_line_num : UDINT; (*Interpeter block monitor: current line number *)
		cur_block_num : UDINT; (*Interpeter block monitor: current line N-block number *)
		intern1 : UDINT; (*[INTERNAL] *)
		intern2 : UDINT; (*[INTERNAL] *)
		intern3 : UDINT; (*[INTERNAL] *)
		intern4 : UDINT; (*[INTERNAL] *)
		intern5 : UDINT; (*[INTERNAL] *)
		breakpoint_count : UDINT; (*Number of breakpoints set *)
		ipvar_access_count : UDINT; (*Number of IP variables being directly accessed by PLC *)
		intern6 : UDINT; (*[INTERNAL] *)
		intern7 : UDINT; (*[INTERNAL] *)
		num_parallel_events : UDINT; (*Number of cyclic jobs currently active *)
		parallel_cycle_count : UDINT; (*Number of execution cycles of all cyclic jobs *)
		parallel_action_text : ARRAY[0..11,0..79]OF USINT; (*cyclic execution monitor - cyclic job source line text *)
		parallel_eval_count : ARRAY[0..11]OF UDINT; (*number of times the cyclic job has been evaluated (tested) *)
		parallel_exec_count : ARRAY[0..11]OF UDINT; (*number of times a Synchronised Action has executed (not relevant to FUBs) *)
		num_fubs_exec_ipsynch : UDINT; (*Number of interpreter synchronous FUBs executing *)
		num_fubs_exec_ppsynch : UDINT; (*Number of path synchronous FUBs executing *)
		callstack : ARRAY[0..11,0..79]OF USINT; (*Program callstack *)
		shared_mem_size : UDINT; (*Memory consumed by shared library data (partitions will be larger) *)
		ip_mem_size : UDINT; (*Memory consumed by interpreter instance (partitions will be larger) *)
		ip_cur_file_mem_size : UDINT; (*Memory consumed by start program (or last loaded program) file (partitions will be larger) *)
		sys_free_mem : UDINT; (*Available system memory *)
		intern8 : UDINT; (*[INTERNAL] *)
		intern9 : UDINT; (*[INTERNAL] *)
		intern10 : UDINT; (*[INTERNAL] *)
		intern11 : UDINT; (*[INTERNAL] *)
		parallel_enabled : USINT; (*Bool: cyclic execution enabled *)
		parallel_rdisable_set : USINT; (*Bool: cyclic jobs set the keep-alive (rdisable) flag *)
		intern12 : USINT; (*[INTERNAL] *)
		intern13 : USINT; (*[INTERNAL] *)
		cur_prog_file_name : ARRAY[0..79]OF USINT; (*File name of the current program*)
		cur_prog_name : ARRAY[0..79]OF USINT; (*Name of the current program*)
	END_STRUCT;
END_TYPE
```

### Optimizer.var - Global variables
```iecst
(********************************************************************
 * COPYRIGHT -- Microsoft
 ********************************************************************
 * Package: Optimizer
 * File: Optimizer.var
 * Author: renj
 * Created: April 24, 2015
 ********************************************************************
 * Variables of package Optimizer
 ********************************************************************)
VAR
	OptMotConfig : OPTMOT_CONFIG_ADVANCED_typ;
END_VAR
```

### Program Logical/MotionHandling/Optimizer/OptMotion (ANSIC)

#### OptMotion.c - Implementation code
```c
/********************************************************************
 * COPYRIGHT -- Bernecker + Rainer
 ********************************************************************
 * Program: OptMotion
 * File: OptMotion.c
 * Author: grubere
 * Created: June 01, 2010
 ********************************************************************
 * Implementation of program OptMotion
 ********************************************************************/

#include <bur/plctypes.h>

#ifdef _DEFAULT_INCLUDES
 #include <AsDefault.h>
#endif

#define PI 3.14159265

void _INIT OptMotionINIT( void )
{
/* ======== Units in [rad], [kg], [m] ======== */

	/* ======== Baseparameter for dynamic model ======== */

	Par6axATrf[0].base_param1 = 0.000000;
	Par6axATrf[0].base_param2 = 0.000000;
	Par6axATrf[0].base_param3 = 0.000000;
	Par6axATrf[0].base_param4 = 0.000000;
	Par6axATrf[0].base_param5 = 0.000000;
	Par6axATrf[0].base_param6 = 0.000000;
	Par6axATrf[0].base_param7 = 0.000000;
	Par6axATrf[0].base_param8 = 71.983100;
	Par6axATrf[0].base_param9 = 0.000000;
	Par6axATrf[0].base_param10 = 0.000000;
	Par6axATrf[0].base_param11 = 0.000000;
	Par6axATrf[0].base_param12 = 0.000000;
	Par6axATrf[0].base_param13 = 0.000000;
	Par6axATrf[0].base_param14 = 0.000000;
	Par6axATrf[0].base_param15 = 0.000000;
	Par6axATrf[0].base_param16 = -0.469116;
	Par6axATrf[0].base_param17 = 0.000000;
	Par6axATrf[0].base_param18 = 21.356410;
	Par6axATrf[0].base_param19 = -7.126585;
	Par6axATrf[0].base_param20 = -1.513853;
	Par6axATrf[0].base_param21 = 0.987800;
	Par6axATrf[0].base_param22 = 0.256704;
	Par6axATrf[0].base_param23 = 0.000000;
	Par6axATrf[0].base_param24 = 26.658310;
	Par6axATrf[0].base_param25 = 0.000000;
	Par6axATrf[0].base_param26 = 0.000000;
	Par6axATrf[0].base_param27 = 0.000000;
	Par6axATrf[0].base_param28 = 0.000000;
	Par6axATrf[0].base_param29 = 0.000000;
	Par6axATrf[0].base_param30 = 9.741126;
	Par6axATrf[0].base_param31 = 0.000000;
	Par6axATrf[0].base_param32 = -0.064780;
	Par6axATrf[0].base_param33 = -5.490367;
	Par6axATrf[0].base_param34 = 2.568725;
	Par6axATrf[0].base_param35 = -2.032787;
	Par6axATrf[0].base_param36 = 6.458844;
	Par6axATrf[0].base_param37 = 0.000000;
	Par6axATrf[0].base_param38 = 2.981729;
	Par6axATrf[0].base_param39 = 0.000000;
	Par6axATrf[0].base_param40 = 0.000000;
	Par6axATrf[0].base_param41 = 0.000000;
	Par6axATrf[0].base_param42 = 0.000000;
	Par6axATrf[0].base_param43 = 0.000000;
	Par6axATrf[0].base_param44 = 0.000000;
	Par6axATrf[0].base_param45 = -0.481579;
	Par6axATrf[0].base_param46 = 0.382556;
	Par6axATrf[0].base_param47 = -0.772865;
	Par6axATrf[0].base_param48 = 0.234084;
	Par6axATrf[0].base_param49 = 1.289617;
	Par6axATrf[0].base_param50 = 0.000000;
	Par6axATrf[0].base_param51 = 1.014531;
	Par6axATrf[0].base_param52 = 3.947117;
	Par6axATrf[0].base_param53 = 0.000000;
	Par6axATrf[0].base_param54 = 0.000000;
	Par6axATrf[0].base_param55 = 0.000000;
	Par6axATrf[0].base_param56 = 0.000000;
	Par6axATrf[0].base_param57 = 0.000000;
	Par6axATrf[0].base_param58 = 1.674332;
	Par6axATrf[0].base_param59 = 0.000000;
	Par6axATrf[0].base_param60 = 0.099178;
	Par6axATrf[0].base_param61 = 0.705105;
	Par6axATrf[0].base_param62 = 0.213770;
	Par6axATrf[0].base_param63 = -0.109433;
	Par6axATrf[0].base_param64 = 1.254646;
	Par6axATrf[0].base_param65 = 0.000000;
	Par6axATrf[0].base_param66 = 0.465107;
	Par6axATrf[0].base_param67 = 0.000000;
	Par6axATrf[0].base_param68 = 0.000000;
	Par6axATrf[0].base_param69 = 0.000000;
	Par6axATrf[0].base_param70 = 0.000000;
	Par6axATrf[0].base_param71 = 0.000000;
	Par6axATrf[0].base_param72 = 0.000000;
	Par6axATrf[0].base_param73 = -0.037241;
	Par6axATrf[0].base_param74 = -0.029525;
	Par6axATrf[0].base_param75 = -0.194226;
	Par6axATrf[0].base_param76 = 0.010846;
	Par6axATrf[0].base_param77 = -0.003949;
	Par6axATrf[0].base_param78 = 0.000000;
	Par6axATrf[0].base_param79 = -0.150153;
	Par6axATrf[0].base_param80 = 0.103083;
	Par6axATrf[0].base_param81 = 0.000000;
	Par6axATrf[0].base_param82 = 0.000000;
	Par6axATrf[0].base_param83 = 0.000000;
	Par6axATrf[0].base_param84 = 0.000000;
	Par6axATrf[0].base_param85 = 0.000000;
	Par6axATrf[0].base_param86 = 0.000000;
	Par6axATrf[0].base_param87 = 0.000000;
	Par6axATrf[0].base_param88 = 0.000000;
	Par6axATrf[0].base_param89 = 0.000000;
	Par6axATrf[0].base_param90 = 0.000000;
	Par6axATrf[0].base_param91 = 0.000000;
	Par6axATrf[0].base_param92 = 0.000000;
	Par6axATrf[0].base_param93 = 0.000000;
	Par6axATrf[0].base_param94 = 0.000000;
	Par6axATrf[0].base_param95 = 0.000000;
	Par6axATrf[0].base_param96 = 0.000000;
	Par6axATrf[0].base_param97 = 0.000000;
	Par6axATrf[0].base_param98 = 470.100069;
	Par6axATrf[0].base_param99 = 43.620507;
	Par6axATrf[0].base_param100 = 16.966225;
	Par6axATrf[0].base_param101 = 47.740884;
	Par6axATrf[0].base_param102 = 3.974347;
	Par6axATrf[0].base_param103 = 1.926903;
	Par6axATrf[0].base_param104 = 234.410106;
	Par6axATrf[0].base_param105 = 28.334038;
	Par6axATrf[0].base_param106 = 24.160627;
	Par6axATrf[0].base_param107 = 48.112117;
	Par6axATrf[0].base_param108 = 9.985319;
	Par6axATrf[0].base_param109 = 5.056168;
	/* ================================== */

	/* ======== Static Parameter ======== */
	Par6axATrf[0].a0x = 0;
	Par6axATrf[0].a0y = 0;
	Par6axATrf[0].a0z = 0;
	Par6axATrf[0].a1x = 0.17;
	Par6axATrf[0].a1y = 0.1415;
	Par6axATrf[0].a1z = 0.45;
	Par6axATrf[0].a2x = 0;
	Par6axATrf[0].a2y = 0;
	Par6axATrf[0].a2z = 0.55;
	Par6axATrf[0].a3x = 0.1775;
	Par6axATrf[0].a3y = -0.1415;
	Par6axATrf[0].a3z = 0.09;
	Par6axATrf[0].a4x = 0.4225;
	Par6axATrf[0].a5x = 0.1;
	Par6axATrf[0].iG1 = 147.5;
	Par6axATrf[0].iG2 = 89;
	Par6axATrf[0].iG3 = 89;
	Par6axATrf[0].iG4 = 160.0;
	Par6axATrf[0].iG5 = 67.74;
	Par6axATrf[0].iG6 = 50;
	Par6axATrf[0].g = 9.81;
	/* ================================== */

/* ======== ax-definition of joint axes ======== */

	OptMotConfig.axes.ax_count = 6;
	OptMotConfig.axes.ax_index[0] = 6;
	OptMotConfig.axes.ax_index[1] = 7;
	OptMotConfig.axes.ax_index[2] = 8;
	OptMotConfig.axes.ax_index[3] = 9;
	OptMotConfig.axes.ax_index[4] = 10;
	OptMotConfig.axes.ax_index[5] = 11;
	OptMotConfig.axes.ax_factor[0] = PI/180.0;
	OptMotConfig.axes.ax_factor[1] = PI/180.0;
	OptMotConfig.axes.ax_factor[2] = PI/180.0;
	OptMotConfig.axes.ax_factor[3] = PI/180.0;
	OptMotConfig.axes.ax_factor[4] = PI/180.0;
	OptMotConfig.axes.ax_factor[5] = PI/180.0;

/* =================== dynamic limits for joint axes =================== */

	OptMotConfig.limits[0].v_joint_max[0] = 95 * OptMotConfig.axes.ax_factor[0];
	OptMotConfig.limits[0].v_joint_max[1] = 90 * OptMotConfig.axes.ax_factor[1];
	OptMotConfig.limits[0].v_joint_max[2] = 90 * OptMotConfig.axes.ax_factor[2];
	OptMotConfig.limits[0].v_joint_max[3] = 120 * OptMotConfig.axes.ax_factor[3];
	OptMotConfig.limits[0].v_joint_max[4] = 120 * OptMotConfig.axes.ax_factor[4];
	OptMotConfig.limits[0].v_joint_max[5] = 190 * OptMotConfig.axes.ax_factor[5];
	OptMotConfig.limits[0].v_joint_min[0] = -OptMotConfig.limits[0].v_joint_max[0];
	OptMotConfig.limits[0].v_joint_min[1] = -OptMotConfig.limits[0].v_joint_max[1];
	OptMotConfig.limits[0].v_joint_min[2] = -OptMotConfig.limits[0].v_joint_max[2];
	OptMotConfig.limits[0].v_joint_min[3] = -OptMotConfig.limits[0].v_joint_max[3];
	OptMotConfig.limits[0].v_joint_min[4] = -OptMotConfig.limits[0].v_joint_max[4];
	OptMotConfig.limits[0].v_joint_min[5] = -OptMotConfig.limits[0].v_joint_max[5];

	OptMotConfig.limits[0].a_joint_max[0] = 5 * OptMotConfig.limits[0].v_joint_max[0];
	OptMotConfig.limits[0].a_joint_max[1] = 5 * OptMotConfig.limits[0].v_joint_max[1];
	OptMotConfig.limits[0].a_joint_max[2] = 5 * OptMotConfig.limits[0].v_joint_max[2];
	OptMotConfig.limits[0].a_joint_max[3] = 5 * OptMotConfig.limits[0].v_joint_max[3];
	OptMotConfig.limits[0].a_joint_max[4] = 5 * OptMotConfig.limits[0].v_joint_max[4];
	OptMotConfig.limits[0].a_joint_max[5] = 5 * OptMotConfig.limits[0].v_joint_max[5];
	OptMotConfig.limits[0].a_joint_min[0] = -OptMotConfig.limits[0].a_joint_max[0];
	OptMotConfig.limits[0].a_joint_min[1] = -OptMotConfig.limits[0].a_joint_max[1];
	OptMotConfig.limits[0].a_joint_min[2] = -OptMotConfig.limits[0].a_joint_max[2];
	OptMotConfig.limits[0].a_joint_min[3] = -OptMotConfig.limits[0].a_joint_max[3];
	OptMotConfig.limits[0].a_joint_min[4] = -OptMotConfig.limits[0].a_joint_max[4];
	OptMotConfig.limits[0].a_joint_min[5] = -OptMotConfig.limits[0].a_joint_max[5];

	OptMotConfig.limits[0].j_joint_max[0] = 20 * OptMotConfig.limits[0].a_joint_max[0];
	OptMotConfig.limits[0].j_joint_max[1] = 40 * OptMotConfig.limits[0].a_joint_max[1];
	OptMotConfig.limits[0].j_joint_max[2] = 40 * OptMotConfig.limits[0].a_joint_max[2];
	OptMotConfig.limits[0].j_joint_max[3] = 40 * OptMotConfig.limits[0].a_joint_max[3];
	OptMotConfig.limits[0].j_joint_max[4] = 40 * OptMotConfig.limits[0].a_joint_max[4];
	OptMotConfig.limits[0].j_joint_max[5] = 40 * OptMotConfig.limits[0].a_joint_max[5];
	OptMotConfig.limits[0].j_joint_min[0] = -OptMotConfig.limits[0].j_joint_max[0];
	OptMotConfig.limits[0].j_joint_min[1] = -OptMotConfig.limits[0].j_joint_max[1];
	OptMotConfig.limits[0].j_joint_min[2] = -OptMotConfig.limits[0].j_joint_max[2];
	OptMotConfig.limits[0].j_joint_min[3] = -OptMotConfig.limits[0].j_joint_max[3];
	OptMotConfig.limits[0].j_joint_min[4] = -OptMotConfig.limits[0].j_joint_max[4];
	OptMotConfig.limits[0].j_joint_min[5] = -OptMotConfig.limits[0].j_joint_max[5];

	OptMotConfig.limits[0].torque_max[0] = 50.5;
	OptMotConfig.limits[0].torque_max[1] = 70.4;
	OptMotConfig.limits[0].torque_max[2] = 30.42;
	OptMotConfig.limits[0].torque_max[3] = 10.35;
	OptMotConfig.limits[0].torque_max[4] = 11.68;
	OptMotConfig.limits[0].torque_max[5] = 11.68;
	OptMotConfig.limits[0].torque_min[0] = -OptMotConfig.limits[0].torque_max[0];
	OptMotConfig.limits[0].torque_min[1] = -OptMotConfig.limits[0].torque_max[1];
	OptMotConfig.limits[0].torque_min[2] = -OptMotConfig.limits[0].torque_max[2];
	OptMotConfig.limits[0].torque_min[3] = -OptMotConfig.limits[0].torque_max[3];
	OptMotConfig.limits[0].torque_min[4] = -OptMotConfig.limits[0].torque_max[4];
	OptMotConfig.limits[0].torque_min[5] = -OptMotConfig.limits[0].torque_max[5];

	/* Limits for path definition 0 */
	OptMotConfig.limits[0].v_path_max[0] = 4000;
	OptMotConfig.limits[0].v_path_min[0] = -4000;
	OptMotConfig.limits[0].a_path_max[0] = 100000;
	OptMotConfig.limits[0].a_path_min[0] = -OptMotConfig.limits[0].a_path_max[0];
	OptMotConfig.limits[0].j_path_max[0] = 500000;
	OptMotConfig.limits[0].j_path_min[0] = -OptMotConfig.limits[0].j_path_max[0];

	/* Limits for path definition 1 */
	OptMotConfig.limits[0].v_path_max[1] = 2000;
	OptMotConfig.limits[0].v_path_min[1] = -2000;
	OptMotConfig.limits[0].a_path_max[1] = 100000;
	OptMotConfig.limits[0].a_path_min[1] = -OptMotConfig.limits[0].a_path_max[0];
	OptMotConfig.limits[0].j_path_max[1] = 1000000;
	OptMotConfig.limits[0].j_path_min[1] = -OptMotConfig.limits[0].j_path_max[0];

	/* Limits for path definition 2 */
	OptMotConfig.limits[0].v_path_max[2] = 2000;
	OptMotConfig.limits[0].v_path_min[2] = -2000;
	OptMotConfig.limits[0].a_path_max[2] = 100000;
	OptMotConfig.limits[0].a_path_min[2] = -OptMotConfig.limits[0].a_path_max[0];
	OptMotConfig.limits[0].j_path_max[2] = 1000000;
	OptMotConfig.limits[0].j_path_min[2] = -OptMotConfig.limits[0].j_path_max[0];

	OptMotConfig.internals.Ts_multiple = 6.0;
	OptMotConfig.internals.buffer_nc_block = 400;
	OptMotConfig.segmentation.distance = 1.0;

	/* =================== path definitions =================== */

	OptMotConfig.path.count = 3;

	// Path definition 0 --> must be used for TRACKING
	// v_path = sqrt( (v_X)^2 + (v_Y)^2 + (v_Z)^2 )
	// Units --> [v_path] = mm/s
	OptMotConfig.path.definition[0].type = 0;
	OptMotConfig.path.definition[0].ax_count = 6;
	OptMotConfig.path.definition[0].ax_index[0] = 0;
	OptMotConfig.path.definition[0].ax_index[1] = 1;
	OptMotConfig.path.definition[0].ax_index[2] = 2;
	OptMotConfig.path.definition[0].ax_index[3] = 3;
	OptMotConfig.path.definition[0].ax_index[4] = 4;
	OptMotConfig.path.definition[0].ax_index[5] = 5;
	OptMotConfig.path.definition[0].ax_factor[0] = 1;
	OptMotConfig.path.definition[0].ax_factor[1] = 1;
	OptMotConfig.path.definition[0].ax_factor[2] = 1;
	OptMotConfig.path.definition[0].ax_factor[3] = 1;
	OptMotConfig.path.definition[0].ax_factor[4] = 1;
	OptMotConfig.path.definition[0].ax_factor[5] = 1;

	// Path definition 1 --> for orientation movements
	// v_path = omega_path = f(v_A, v_B, v_C)
	// Units --> [v_path] = ?s
	OptMotConfig.path.definition[1].type = 1;
	OptMotConfig.path.definition[1].ax_count = 3;
	OptMotConfig.path.definition[1].ax_index[0] = 3;
	OptMotConfig.path.definition[1].ax_index[1] = 4;
	OptMotConfig.path.definition[1].ax_index[2] = 5;
	OptMotConfig.path.definition[1].ax_factor[0] = 1;
	OptMotConfig.path.definition[1].ax_factor[1] = 1;
	OptMotConfig.path.definition[1].ax_factor[2] = 1;

	// Path definition 2 --> for PTP movements
	// v_path = sqrt( (v_Q1)^2 + (v_Q2)^2 + (v_Q3)^2 + (v_Q4)^2 + (v_Q5)^2 + (v_Q6)^2 )
	// Units with ax_factor[] = 1: --> [v_path] = ?s
	OptMotConfig.path.definition[2].type = 0;
	OptMotConfig.path.definition[2].ax_count = 6;
	OptMotConfig.path.definition[2].ax_index[0] = 6;
	OptMotConfig.path.definition[2].ax_index[1] = 7;
	OptMotConfig.path.definition[2].ax_index[2] = 8;
	OptMotConfig.path.definition[2].ax_index[3] = 9;
	OptMotConfig.path.definition[2].ax_index[4] = 10;
	OptMotConfig.path.definition[2].ax_index[5] = 11;
	OptMotConfig.path.definition[2].ax_factor[0] = 1;
	OptMotConfig.path.definition[2].ax_factor[1] = 1;
	OptMotConfig.path.definition[2].ax_factor[2] = 1;
	OptMotConfig.path.definition[2].ax_factor[3] = 1;
	OptMotConfig.path.definition[2].ax_factor[4] = 1;
	OptMotConfig.path.definition[2].ax_factor[5] = 1;

	/* =================== tracking configuration =================== */

	OptMotConfig.path.tracking.enable = 0;
	OptMotConfig.path.tracking.conveyorData.orientationParameter.angles_type = TRF_CARDAN_XYZ_ANGLES;
	OptMotConfig.path.tracking.conveyorData.orientationParameter.measure = TRF_DEGREES;

	//first conveyor
	OptMotConfig.path.tracking.conveyorData.conveyor[0].limits.maxVelocity = 100;
	OptMotConfig.path.tracking.conveyorData.conveyor[0].orientation.phi = 0;
	OptMotConfig.path.tracking.conveyorData.conveyor[0].orientation.theta = 0;
	OptMotConfig.path.tracking.conveyorData.conveyor[0].orientation.psi = 90;

}

void _CYCLIC OptMotionCYCLIC( void )
{

}
```

### Package Logical/HmiHandling - Hmi Handling

### HmiGlobal.typ - Global data types
```iecst
(********************************************************************
 * COPYRIGHT --
 ********************************************************************
 * Package: Hmi
 * File: Hmi.typ
 * Author: liug
 * Created: March 04, 2013
 ********************************************************************
 * Data types of package Hmi
 ********************************************************************)

TYPE
	HmiGlobal_Type : 	STRUCT
		Address : HmiGlobalAddress_Type;
		PageControl : HmiGlobalPageCtrl_Type;
	END_STRUCT;
	HmiGlobalPageCtrl_Type : 	STRUCT
		ActPage : UINT;
		SetPage : UINT;
	END_STRUCT;
	HmiGlobalAddress_Type : 	STRUCT
		SystemAddress : UDINT;
		AxesAddress : UDINT;
		CncAddress : UDINT;
		JogAddress : UDINT;
		RecipeAddress : UDINT;
		ErrorAddress : UDINT;
	END_STRUCT;
	HmiEditControl_Type : 	STRUCT
		CommandRequest : STRING[200];
		CommandResponse : STRING[200];
		CommandStatus : UINT;
		CursorLine : UDINT;
		StatusDatapoint : UINT;
		LastExcuteLine : DINT;
		LastHighLightLine : DINT;
		URL : STRING[80];
		CursorCol : UDINT;
		TargetCursorCol : UDINT;
		TargetCursorLine : UDINT;
	END_STRUCT;
	HmiRetain_Type : 	STRUCT
		HmiProgram : HmiProgramRetain_Type;
		HmiKeyControl : HmiKeyControlRetain_Type;
		HmiEditor : HmiEditorRetain_Type;
		HmiRobot : HmiRobot_Type;
		HmiJog : HmiJogRetain_Type;
	END_STRUCT;
	HmiJogToolRetainType : 	STRUCT
		VarName : STRING[30];
		Tool : MXToolType;
	END_STRUCT;
	HmiJogJointRetainType : 	STRUCT
		VarName : STRING[30];
		Joint : MXAxisTargetType;
		Set : BOOL;
	END_STRUCT;
	HmiJogPointRetainType : 	STRUCT
		VarName : STRING[30];
		Point : {REDUND_UNREPLICABLE} MXPointType;
		Set : BOOL;
	END_STRUCT;
	HmiJogFrameRetainType : 	STRUCT
		VarName : STRING[30];
		Frame : MXFrameType;
	END_STRUCT;
	HmiJogRetain_Type : 	STRUCT
		Frame : HmiJogFrameRetainType;
		Tool : HmiJogToolRetainType;
		Joint : HmiJogJointRetainType;
		Point : HmiJogPointRetainType;
		Name : STRING[80];
		Device : STRING[80];
	END_STRUCT;
	HmiCartesianLimitType : 	STRUCT
		Min : REAL;
		Max : REAL;
	END_STRUCT;
	HmiJointLimitType : 	STRUCT
		Max : REAL;
		Min : REAL;
	END_STRUCT;
	HmiMechType : 	STRUCT
		OffsetY : REAL;
		OffsetZ : REAL;
		OffsetX : REAL;
		Direction : USINT;
	END_STRUCT;
	HmiCouplingType : 	STRUCT
		Coefficient : LREAL;
		Enable : BOOL;
	END_STRUCT;
	HmiRobot_Type : 	STRUCT
		JointLimits : ARRAY[0..5]OF HmiJointLimitType;
		CartesianLimits : ARRAY[0..2]OF HmiCartesianLimitType;
		HomePos : MXPointType;
		Mech : ARRAY[0..5]OF HmiMechType;
		Coupling : ARRAY[0..2]OF HmiCouplingType; (*0: 4->5 1:5->6 2:4-6*)
	END_STRUCT;
	HmiKeyControlRetain_Type : 	STRUCT
		MechHomeOK : BOOL;
	END_STRUCT;
	HmiEditorRetain_Type : 	STRUCT
		Name : STRING[80];
		URLPathOnly : STRING[80];
		URL : STRING[80];
		Device : STRING[80];
	END_STRUCT;
	HmiProgramRetain_Type : 	STRUCT
		Name : STRING[80];
		Mode : USINT;
		URLPathOnly : STRING[80];
		URL : STRING[80];
		Device : STRING[80];
		Ptr : UINT;
	END_STRUCT;
	HmiFileCtrlOutputStatus_Type : 	STRUCT
		ReadOK : BOOL;
		WriteOK : BOOL;
		Busy : BOOL;
	END_STRUCT;
	HmiFileCtrlOutput_Type : 	STRUCT
		Status : HmiFileCtrlOutputStatus_Type;
	END_STRUCT;
	HmiFileCtrlInputCmd_Type : 	STRUCT
		Read : BOOL;
		Write : BOOL;
		AckError : BOOL;
	END_STRUCT;
	HmiFileCtrlInputParam_Type : 	STRUCT
		FileName : STRING[80];
		StringBufferSize : UDINT;
		StringBufferAdr : UDINT;
		FileDevice : STRING[80];
	END_STRUCT;
	HmiFileCtrlInput_Type : 	STRUCT
		Command : HmiFileCtrlInputCmd_Type;
		Parameter : HmiFileCtrlInputParam_Type;
	END_STRUCT;
	HmiFileCtrl_Type : 	STRUCT
		Input : HmiFileCtrlInput_Type;
		Output : HmiFileCtrlOutput_Type;
	END_STRUCT;
END_TYPE

(*VisualComponentsType*)

TYPE
	HmiButtonType : 	STRUCT
		Value : USINT;
		OldValue : USINT;
		StatusDatapoint : UINT;
		CompletionDatapoint : USINT;
		BmpIdx : USINT;
	END_STRUCT;
	HmiLayerType : 	STRUCT
		StatusDatapoint : UINT;
	END_STRUCT;
	HmiScaleType : 	STRUCT
		StartDatapoint : REAL;
		EndDatapoint : REAL;
	END_STRUCT;
	HmiSliderType : 	STRUCT
		Value : REAL;
		StatusDatapoint : UINT;
	END_STRUCT;
	HmiStringType : 	STRUCT
		Value : STRING[80];
		StatusDatapoint : UINT;
	END_STRUCT;
	HmiNumericTypeR : 	STRUCT
		Value : REFERENCE TO REAL;
		StatusDatapoint : UINT;
	END_STRUCT;
	HmiDropdownTypeR : 	STRUCT
		SelectedIndex : REFERENCE TO USINT;
		OldIndex : USINT;
	END_STRUCT;
	HmiNumericType : 	STRUCT
		Value : REAL;
		StatusDatapoint : UINT;
	END_STRUCT;
	HmiTextType : 	STRUCT
		TextIndex : USINT;
		StatusDatapoint : UINT;
	END_STRUCT;
	HmiEditType : 	STRUCT
		CommandRequest : STRING[200];
		CommandResponse : STRING[200];
		CommandStatus : UINT;
		CursorLine : UDINT;
		CursorCol : UDINT;
		URL : STRING[80];
		StatusDatapoint : UINT;
		StringBuffer : STRING[10000];
	END_STRUCT;
	HmiDropdownType : 	STRUCT
		SelectedIndex : USINT;
		OldIndex : USINT;
	END_STRUCT;
	HmiHotSpotType : 	STRUCT
		Value : USINT;
		OldValue : USINT;
	END_STRUCT;
	HmiListboxType : 	STRUCT
		Entries : ARRAY[0..19]OF STRING[80];
		MaxListIndex : USINT;
		SelectedIndex : USINT;
		CompletionDatapoint : USINT;
		OldSelectedIndex : USINT;
		IsEmpty : BOOL;
	END_STRUCT;
	HmiTabsType : 	STRUCT
		TabMaxIndex : USINT;
		TabSelectedIndex : USINT;
		ButtonsTab : ARRAY[0..4]OF HmiButtonType;
		TabBg : HmiTextType;
	END_STRUCT;
	HmiPopupType : 	STRUCT
		Layer : HmiLayerType;
		ButtonCancel : HmiButtonType;
		ButtonConfirm : HmiButtonType;
	END_STRUCT;
	HmiNumericWithRangeType : 	STRUCT
		Value : REAL;
		StatusDatapoint : UINT;
		Max : REAL;
		Min : REAL;
	END_STRUCT;
	HmiBitmapType : 	STRUCT
		BmpIndex : USINT;
	END_STRUCT;
	HmiPopupWithStringType : 	STRUCT
		Layer : HmiLayerType;
		ButtonCancel : HmiButtonType;
		ButtonConfirm : HmiButtonType;
		StringInput : HmiStringType;
		TextInfo : HmiTextType;
	END_STRUCT;
	HmiSimpleType : 	STRUCT
		StatusDatapoint : UINT;
	END_STRUCT;
END_TYPE
```

### HmiGlobal.var - Global variables
```iecst
(********************************************************************
 * COPYRIGHT --
 ********************************************************************
 * Package: Hmi
 * File: Hmi.var
 * Author: liug
 * Created: March 04, 2013
 ********************************************************************
 * Variables of package Hmi
 ********************************************************************)
VAR
	MX_POINT_ZERO : {REDUND_UNREPLICABLE} MXPointType := (0);
	MX_FRAME_ZERO : {REDUND_UNREPLICABLE} MXFrameType := (0);
	MX_TOOL_ZERO : {REDUND_UNREPLICABLE} MXToolType := (0);
	HmiGlobal : HmiGlobal_Type;
END_VAR
VAR RETAIN
	HmiRetain : HmiRetain_Type;
END_VAR
(*Global Alarm*)
VAR
	WarnMessage : ARRAY[0..WARN_MESSAGE_NUM] OF BOOL;
END_VAR
(*Constants*)
VAR CONSTANT
	MAX_REAL_AX_MINUS_ONE : USINT := 5;
	ARSIM_PC : USINT := 3;
	MAX_DEVICES : UINT := 9;
	MAX_PLUS_MINUS_KEY : USINT := 6;
	MAX_PLUS_MINUS_KEY_MINUS_ONE : USINT := MAX_PLUS_MINUS_KEY-1;
	MAX_FUNCTION_KEY : USINT := 9;
	MAX_FUNCTION_KEY_MINUS_ONE : USINT := MAX_FUNCTION_KEY-1;
	MAX_PAGE_KEY : USINT := 7;
	MAX_PAGE_KEY_MINUS_ONE : USINT := MAX_PAGE_KEY-1;
	MAX_ERRORS : UINT := 1000; (*maximum number of errors recorded in history*)
	MAX_ALARMS : USINT := 100; (*maximum number of defined alarms*)
	MAX_WARNINGS : USINT := 50; (*maximum number of defined warnings*)
	MAX_FIELD_ALRAMS : USINT := 6; (*maximum number of field alarms*)
	PAGE_MAIN : UINT := 100;
	PAGE_SETUPKINEMATICS : UINT := 230;
	PAGE_SETUPAXIS : UINT := 220;
	PAGE_SETUPCALIB : UINT := 240;
	PAGE_SETUP : UINT := 200;
	PAGE_IO : UINT := 300;
	PAGE_PROGRAM : UINT := 400;
	PAGE_EDITOR : UINT := 500;
	PAGE_EDITOR_DATA : UINT := 510;
	PAGE_JOGGING : UINT := 600;
	PAGE_ALARM : UINT := 700;
	STRING_PER_LINE : USINT := 120;
	PROG_READ_NUMBER : UDINT := STRING_PER_LINE*PROG_CMD_NUMBER;
	PROG_CMD_NUMBER : UINT := 1000;
	LAYER_HIDE : USINT := 1;
	LAYER_SHOW : USINT := 0;
	LANG_ENGLISH : USINT := 0;
	LANG_CHINESE : USINT := 1;
	USER_GUEST : USINT := 0;
	USER_OPERATOR : USINT := 1;
	USER_PROGRAMMER : USINT := 2;
	LINENUMBER_PERPAGE : USINT := 19;
	LINENUMBER_PERPAGE_MINUS : USINT := LINENUMBER_PERPAGE-1;
	WARN_MESSAGE_NUM : USINT := 19;
	USER_ADMINISTRATOR : USINT := 3;
	ERROR : USINT := 3;
	LOCK : USINT := 2;
	AUTO : USINT := 1;
	DISABLED : USINT := 3;
	JOG : USINT := 0;
	RUN : USINT := 2;
	PAUSE : USINT := 1;
	STOP : USINT := 0;
END_VAR
```

### Package Logical/HmiHandling/HmiHardKey - Hard Key On MP50

### HmiHardKeyGlobal.typ - Global data types
```iecst
(********************************************************************
 * COPYRIGHT --
 ********************************************************************
 * Package: HmiHardKey
 * File: HmiHardKeyGlobal.typ
 * Author: renj
 * Created: March 04, 2013
 ********************************************************************
 * Data types of package HmiHardKey
 ********************************************************************)

TYPE
	HmiHardKeyOutput_Typ : 	STRUCT
		Run_Led : USINT;
		Error_Led : USINT;
		Motion_Led : USINT;
		Process_Led : USINT;
		KeyLevel : USINT;
	END_STRUCT;
	HmiHardKeyInput_Typ : 	STRUCT
		MP50_SimKey : ARRAY[0..50]OF BOOL;
		MP50_Key : ARRAY[0..50]OF BOOL;
		Joystick_XValue : DINT;
		Joystick_YValue : DINT;
		Joystick_ZValue : DINT;
	END_STRUCT;
	HmiHardKey_Type : 	STRUCT
		Input : HmiHardKeyInput_Typ;
		Output : HmiHardKeyOutput_Typ;
	END_STRUCT;
END_TYPE
```

### HmiHardKeyGlobal.var - Global variables
```iecst
(********************************************************************
 * COPYRIGHT --
 ********************************************************************
 * Package: HardKey
 * File: HardKeyGlobal.var
 * Author: renj
 * Created: March 04, 2013
 ********************************************************************
 * Variables of package HardKey
 ********************************************************************)
VAR
	HmiHardKey : HmiHardKey_Type := (0);
END_VAR
```

### Program Logical/HmiHandling/HmiHardKey/HmiHardKeyCtrl (ANSIC) - A new program

#### HmiHardKeyCtrl.c - Implementation code
```c
/********************************************************************
 * COPYRIGHT --
 ********************************************************************
 * Program: HardKeySim
 * File: HardKeySim.c
 * Author: Administrator
 * Created: April 23, 2012
 ********************************************************************
 * Implementation of program HardKeySim
 ********************************************************************/

#include <bur/plctypes.h>

#include <AsRfbExt.h>

#ifdef _DEFAULT_INCLUDES
#include <AsDefault.h>
#endif

void _INIT avcINIT(void)
{
	uiTimeOut = 500;
	Status_RfbExtInit = RfbExtInit(&pLib, uiTimeOut);	/*	Initialize RfbExt functions	*/
	Enable_RfbExtConnect = 1;
}

void _CYCLIC avcCYCLIC(void)
{

	if (Enable_RfbExtConnect == 1)
	{
		Status_RfbExtConnect = RfbExtConnect((UDINT)&pLib, (UDINT) "Visu");
		if (!Status_RfbExtConnect)
			Enable_RfbExtConnect = 0;
	}

	Status_RfbExtDataAge = RfbExtDataAge(&pLib, (UDINT)&pAge);

	if (pAge <= uiTimeOut)		/*	Otherwise there is no connection to the B&R VNC viewer	*/
	{
		Status_RfbExtJoystickValue = RfbExtJoystickValue(&pLib, 0, &HmiHardKey.Input.Joystick_YValue, &HmiHardKey.Input.Joystick_XValue, &HmiHardKey.Input.Joystick_ZValue);
	}

}
```

#### HmiHardKeyLocal.var - Local variables
```iecst
(********************************************************************
 * COPYRIGHT --
 ********************************************************************
 * Program: HardKeySim
 * File: HardKeySim.var
 * Author: liug
 * Created: March 04, 2013
 ********************************************************************
 * Local variables of program HardKeySim
 ********************************************************************)
VAR
	Enable_RfbExtConnect : BOOL := FALSE;
	pAge : UDINT := 0;
	Status_RfbExtDataAge : UDINT := 0;
	uiTimeOut : UDINT := 0;
	Status_RfbExtJoystickValue : UINT := 0;
	Status_RfbExtConnect : UINT := 0;
	pLib : AsRfbExtType := (0);
	Status_RfbExtInit : UINT := 0;
END_VAR
```

### Package Logical/HmiHandling/HmiKeyCtrl - Common Control
